i := 0; WHILE i < COUNT_LOGIC_TS DO
	iecDB_ts[ADRBASE_TS_LOGICAL + i].siq.b.SPI := sys_logic_ts[i];
	i := i + 1;
END_WHILE

i := 0; WHILE i < COUNT_VALVE DO
	iecDB_ts[ADRBASE_TS_VALVE + i*14 + 0].siq.b.SPI := sys_valve[i].flags.mode_dist;
	iecDB_ts[ADRBASE_TS_VALVE + i*14 + 1].siq.b.SPI := sys_valve[i].flags.mode_auto;
	iecDB_ts[ADRBASE_TS_VALVE + i*14 + 2].siq.b.SPI := sys_valve[i].flags.mode_imit;
	iecDB_ts[ADRBASE_TS_VALVE + i*14 + 3].siq.b.SPI := sys_valve[i].flags.mode_block;
	iecDB_ts[ADRBASE_TS_VALVE + i*14 + 4].siq.b.SPI := sys_valve[i].flags.cv_ok;
	iecDB_ts[ADRBASE_TS_VALVE + i*14 + 5].siq.b.SPI := sys_valve[i].flags.cv_fail;
	iecDB_ts[ADRBASE_TS_VALVE + i*14 + 6].siq.b.SPI := sys_valve[i].flags.fail_local;
	iecDB_ts[ADRBASE_TS_VALVE + i*14 + 7].siq.b.SPI := sys_valve[i].flags.fail_block;
	iecDB_ts[ADRBASE_TS_VALVE + i*14 + 8].siq.b.SPI := sys_valve[i].flags.fail_sm;
	iecDB_ts[ADRBASE_TS_VALVE + i*14 + 9].siq.b.SPI := sys_valve[i].flags.fail_start_open;
	iecDB_ts[ADRBASE_TS_VALVE + i*14 + 10].siq.b.SPI := sys_valve[i].flags.fail_open;
	iecDB_ts[ADRBASE_TS_VALVE + i*14 + 11].siq.b.SPI := sys_valve[i].flags.fail_start_close;
	iecDB_ts[ADRBASE_TS_VALVE + i*14 + 12].siq.b.SPI := sys_valve[i].flags.fail_close;
	iecDB_ts[ADRBASE_TS_VALVE + i*14 + 13].siq.b.SPI := sys_valve[i].flags.fail_moving;
	i := i + 1;
END_WHILE

i := 0; WHILE i < COUNT_STOP DO
	iecDB_ts[ADRBASE_TS_STOP + i*6 + 0].siq.b.SPI := sys_stop[i].flags.mode_block;
	iecDB_ts[ADRBASE_TS_STOP + i*6 + 1].siq.b.SPI := sys_stop[i].flags.msg_confirm;
	iecDB_ts[ADRBASE_TS_STOP + i*6 + 2].siq.b.SPI := sys_stop[i].flags.executing;
	iecDB_ts[ADRBASE_TS_STOP + i*6 + 3].siq.b.SPI := sys_stop[i].flags.done;
	iecDB_ts[ADRBASE_TS_STOP + i*6 + 4].siq.b.SPI := sys_stop[i].flags.fail;
	iecDB_ts[ADRBASE_TS_STOP + i*6 + 5].siq.b.SPI := sys_stop[i].flags.fail_block;
	i := i + 1;
END_WHILE

i := 0; WHILE i < COUNT_UNIT DO
	iecDB_ts[ADRBASE_TS_UNIT + i*10 + 0].siq.b.SPI := sys_unit[i].flags.mode_dist;
	iecDB_ts[ADRBASE_TS_UNIT + i*10 + 1].siq.b.SPI := sys_unit[i].flags.mode_auto;
	iecDB_ts[ADRBASE_TS_UNIT + i*10 + 2].siq.b.SPI := sys_unit[i].flags.mode_imit;
	iecDB_ts[ADRBASE_TS_UNIT + i*10 + 3].siq.b.SPI := sys_unit[i].flags.mode_block;
	iecDB_ts[ADRBASE_TS_UNIT + i*10 + 4].siq.b.SPI := sys_unit[i].flags.mode_work;
	iecDB_ts[ADRBASE_TS_UNIT + i*10 + 5].siq.b.SPI := sys_unit[i].flags.cv_ok;
	iecDB_ts[ADRBASE_TS_UNIT + i*10 + 6].siq.b.SPI := sys_unit[i].flags.cv_fail;	
	iecDB_ts[ADRBASE_TS_UNIT + i*10 + 7].siq.b.SPI := sys_unit[i].flags.fail_local;
	iecDB_ts[ADRBASE_TS_UNIT + i*10 + 8].siq.b.SPI := sys_unit[i].flags.fail_block;
	iecDB_ts[ADRBASE_TS_UNIT + i*10 + 9].siq.b.SPI := sys_unit[i].flags.fail_switch;
	i := i + 1;
END_WHILE

i := 0; WHILE i < COUNT_FAIL DO
	iecDB_ts[ADRBASE_TS_FAIL + i*3 + 0].siq.b.SPI := sys_fail[i].processed;
	iecDB_ts[ADRBASE_TS_FAIL + i*3 + 1].siq.b.SPI := sys_fail[i].block;
	iecDB_ts[ADRBASE_TS_FAIL + i*3 + 2].siq.b.SPI := sys_fail[i].imit;
	i := i + 1;
END_WHILE

i := 0; WHILE i < COUNT_WARN DO
	iecDB_ts[ADRBASE_TS_WARN + i*3 + 0].siq.b.SPI := sys_warn[i].processed;
	iecDB_ts[ADRBASE_TS_WARN + i*3 + 1].siq.b.SPI := sys_warn[i].block;
	iecDB_ts[ADRBASE_TS_WARN + i*3 + 2].siq.b.SPI := sys_warn[i].imit;
	i := i + 1;
END_WHILE

// ========== IEC_M_ME_TE
i := 0; WHILE i < COUNT_LOGIC_TE DO
	iecDB_te[ADRBASE_TE_LOGICAL + i].value := INT_TO_WORD(sys_logic_te[i]);
	iecDB_te[ADRBASE_TE_LOGICAL + i].qds.value := USINT_TO_BYTE(RLTBIO.Constants.QDS_STT_OK);
	i := i + 1;
END_WHILE

i := 0; WHILE i < COUNT_VALVE DO
	iecDB_te[ADRBASE_TE_VALVE + i*5 + 0].value := INT_TO_WORD(sys_valve[i].v_mode);
	iecDB_te[ADRBASE_TE_VALVE + i*5 + 0].qds.value := USINT_TO_BYTE(RLTBIO.Constants.QDS_STT_OK);
	iecDB_te[ADRBASE_TE_VALVE + i*5 + 1].value := INT_TO_WORD(sys_valve[i].v_state);
	iecDB_te[ADRBASE_TE_VALVE + i*5 + 1].qds.value := USINT_TO_BYTE(RLTBIO.Constants.QDS_STT_OK);
	iecDB_te[ADRBASE_TE_VALVE + i*5 + 2].value := sys_valve[i].sp.start;
	iecDB_te[ADRBASE_TE_VALVE + i*5 + 2].qds.value := USINT_TO_BYTE(RLTBIO.Constants.QDS_STT_OK);
	iecDB_te[ADRBASE_TE_VALVE + i*5 + 3].value := sys_valve[i].sp.moving;
	iecDB_te[ADRBASE_TE_VALVE + i*5 + 3].qds.value := USINT_TO_BYTE(RLTBIO.Constants.QDS_STT_OK);
	iecDB_te[ADRBASE_TE_VALVE + i*5 + 4].value := sys_valve[i].sp.press;
	iecDB_te[ADRBASE_TE_VALVE + i*5 + 4].qds.value := USINT_TO_BYTE(RLTBIO.Constants.QDS_STT_OK);
	i := i + 1;
END_WHILE

i := 0; WHILE i < COUNT_STOP DO
	iecDB_te[ADRBASE_TE_STOP + i*2 + 0].value := INT_TO_WORD(sys_stop[i].status);
	iecDB_te[ADRBASE_TE_STOP + i*2 + 0].qds.value := USINT_TO_BYTE(RLTBIO.Constants.QDS_STT_OK);
	iecDB_te[ADRBASE_TE_STOP + i*2 + 1].value := sys_stop[i].step;
	iecDB_te[ADRBASE_TE_STOP + i*2 + 1].qds.value := USINT_TO_BYTE(RLTBIO.Constants.QDS_STT_OK);
	i := i + 1;
END_WHILE

i := 0; WHILE i < COUNT_UNIT DO
	iecDB_te[ADRBASE_TE_UNIT + i*2 + 0].value := sys_unit[i].sp.switch;
	iecDB_te[ADRBASE_TE_UNIT + i*2 + 0].qds.value := USINT_TO_BYTE(RLTBIO.Constants.QDS_STT_OK);
	iecDB_te[ADRBASE_TE_UNIT + i*2 + 1].value := sys_unit[i].sp.work;
	iecDB_te[ADRBASE_TE_UNIT + i*2 + 1].qds.value := USINT_TO_BYTE(RLTBIO.Constants.QDS_STT_OK);
	i := i + 1;
END_WHILE

// ========== IEC_M_ME_TF
i := 0; WHILE i < COUNT_LOGIC_TF DO
	iecDB_tf[ADRBASE_TF_LOGICAL + i].value := sys_logic_tf[i];
	iecDB_tf[ADRBASE_TF_LOGICAL + i].qds.value := USINT_TO_BYTE(RLTBIO.Constants.QDS_STT_OK);
	i := i + 1;
END_WHILE

i := 0; WHILE i < COUNT_AI DO
	iecDB_tf[ADRBASE_TF_TI_VALUE + i*9 + 0].value := sys_ai[i].rTI;
	iecDB_tf[ADRBASE_TF_TI_VALUE + i*9 + 0].qds.value := USINT_TO_BYTE(sys_ai[i].qds);
	iecDB_tf[ADRBASE_TF_TI_VALUE + i*9 + 1].value := sys_ai[i].out_min;
	iecDB_tf[ADRBASE_TF_TI_VALUE + i*9 + 1].qds.value := USINT_TO_BYTE(RLTBIO.Constants.QDS_STT_OK);
	iecDB_tf[ADRBASE_TF_TI_VALUE + i*9 + 2].value := sys_ai[i].out_max;
	iecDB_tf[ADRBASE_TF_TI_VALUE + i*9 + 2].qds.value := USINT_TO_BYTE(RLTBIO.Constants.QDS_STT_OK);
	iecDB_tf[ADRBASE_TF_TI_VALUE + i*9 + 3].value := sys_ai[i].delta;
	iecDB_tf[ADRBASE_TF_TI_VALUE + i*9 + 3].qds.value := USINT_TO_BYTE(RLTBIO.Constants.QDS_STT_OK);
	iecDB_tf[ADRBASE_TF_TI_VALUE + i*9 + 4].value := sys_ai[i].val_fail_min;
	iecDB_tf[ADRBASE_TF_TI_VALUE + i*9 + 4].qds.value := USINT_TO_BYTE(RLTBIO.Constants.QDS_STT_OK);
	iecDB_tf[ADRBASE_TF_TI_VALUE + i*9 + 5].value := sys_ai[i].val_fail_max;
	iecDB_tf[ADRBASE_TF_TI_VALUE + i*9 + 5].qds.value := USINT_TO_BYTE(RLTBIO.Constants.QDS_STT_OK);
	iecDB_tf[ADRBASE_TF_TI_VALUE + i*9 + 6].value := sys_ai[i].val_warn_min;
	iecDB_tf[ADRBASE_TF_TI_VALUE + i*9 + 6].qds.value := USINT_TO_BYTE(RLTBIO.Constants.QDS_STT_OK);
	iecDB_tf[ADRBASE_TF_TI_VALUE + i*9 + 7].value := sys_ai[i].val_warn_max;
	iecDB_tf[ADRBASE_TF_TI_VALUE + i*9 + 7].qds.value := USINT_TO_BYTE(RLTBIO.Constants.QDS_STT_OK);
	iecDB_tf[ADRBASE_TF_TI_VALUE + i*9 + 8].value := sys_ai[i].hyst;
	iecDB_tf[ADRBASE_TF_TI_VALUE + i*9 + 8].qds.value := USINT_TO_BYTE(RLTBIO.Constants.QDS_STT_OK);
	i := i + 1;
END_WHILE

i := 0; WHILE i < COUNT_AO DO
	iecDB_tf[ADRBASE_TF_TR_VALUE + i*3 + 0].value := sys_ao[i].tr;
	iecDB_tf[ADRBASE_TF_TR_VALUE + i*3 + 0].qds.value := USINT_TO_BYTE(RLTBIO.Constants.QDS_STT_OK);
	iecDB_tf[ADRBASE_TF_TR_VALUE + i*3 + 1].value := sys_ao[i].in_min;
	iecDB_tf[ADRBASE_TF_TR_VALUE + i*3 + 1].qds.value := USINT_TO_BYTE(RLTBIO.Constants.QDS_STT_OK);
	iecDB_tf[ADRBASE_TF_TR_VALUE + i*3 + 2].value := sys_ao[i].in_max;
	iecDB_tf[ADRBASE_TF_TR_VALUE + i*3 + 2].qds.value := USINT_TO_BYTE(RLTBIO.Constants.QDS_STT_OK);
	i := i + 1;
END_WHILE

//========== C_SC_NA_1		через ИЛИ потому что могут быть и другие источники команд!
station.cmd.mode_auto_off := station.cmd.mode_auto_off OR		iecDB_tu[1];	iecDB_tu[1] := FALSE;
station.cmd.mode_auto_on := station.cmd.mode_auto_on OR			iecDB_tu[2];	iecDB_tu[2] := FALSE;
station.cmd.ack_control := station.cmd.ack_control OR			iecDB_tu[3];	iecDB_tu[3] := FALSE;
station.cmd.ack_valves := station.cmd.ack_valves OR				iecDB_tu[4];	iecDB_tu[4] := FALSE;
station.cmd.ack_units := station.cmd.ack_units OR				iecDB_tu[5];	iecDB_tu[5] := FALSE;
station.cmd.ack_alarms := station.cmd.ack_alarms OR				iecDB_tu[6];	iecDB_tu[6] := FALSE;
station.cmd.reset_imit := station.cmd.reset_imit OR 			iecDB_tu[7];	iecDB_tu[7] := FALSE;
station.cmd.imit_valves_on := station.cmd.imit_valves_on OR 	iecDB_tu[8];	iecDB_tu[8] := FALSE;
station.cmd.imit_valves_off := station.cmd.imit_valves_off OR	iecDB_tu[9];	iecDB_tu[9] := FALSE;
station.cmd.imit_units_on := station.cmd.imit_units_on OR		iecDB_tu[10];	iecDB_tu[10] := FALSE;
station.cmd.imit_units_off := station.cmd.imit_units_off OR		iecDB_tu[11];	iecDB_tu[11] := FALSE;
station.cmd.block_sound_on := station.cmd.block_sound_on OR		iecDB_tu[12];	iecDB_tu[12] := FALSE;
station.cmd.block_sound_off := station.cmd.block_sound_off OR	iecDB_tu[13];	iecDB_tu[13] := FALSE;
station.cmd.sound_on := station.cmd.sound_on OR					iecDB_tu[14];	iecDB_tu[14] := FALSE;
station.cmd.sound_off := station.cmd.sound_off OR				iecDB_tu[15];	iecDB_tu[15] := FALSE;
station.cmd.alarm_on := station.cmd.alarm_on OR					iecDB_tu[16];	iecDB_tu[16] := FALSE;
station.cmd.alarm_off := station.cmd.alarm_off OR				iecDB_tu[17];	iecDB_tu[17] := FALSE;
station.cmd.lamps_on := station.cmd.lamps_on OR 				iecDB_tu[18];	iecDB_tu[18] := FALSE;
station.cmd.lamps_off := station.cmd.lamps_off OR 				iecDB_tu[19];	iecDB_tu[19] := FALSE;
//i := 0; WHILE i < COUNT_LOGIC_CMD DO
//	iecDB_tu[ADRBASE_CMD_LOGIC + i] := FALSE;
//	i := i + 1;
//END_WHILE

i := 0; WHILE i < COUNT_VALVE DO
	IF station.mode <> en_stt_mode.MODE_AUTO THEN
		sys_valve[i].cmd.open := sys_valve[i].cmd.open OR			iecDB_tu[ADRBASE_CMD_VALVE + i*8 + 0];
		sys_valve[i].cmd.close := sys_valve[i].cmd.close OR			iecDB_tu[ADRBASE_CMD_VALVE + i*8 + 1];
		sys_valve[i].cmd.stop := sys_valve[i].cmd.stop OR			iecDB_tu[ADRBASE_CMD_VALVE + i*8 + 2];
	ELSE
		IF sys_valve[i].cmd.open OR sys_valve[i].cmd.close OR sys_valve[i].cmd.stop THEN
			station.fail_control := TRUE;
		END_IF
	END_IF
	iecDB_tu[ADRBASE_CMD_VALVE + i*8 + 0] := FALSE;
	iecDB_tu[ADRBASE_CMD_VALVE + i*8 + 1] := FALSE;
	iecDB_tu[ADRBASE_CMD_VALVE + i*8 + 2] := FALSE;
	sys_valve[i].cmd.ack := sys_valve[i].cmd.ack OR				iecDB_tu[ADRBASE_CMD_VALVE + i*8 + 3];		iecDB_tu[ADRBASE_CMD_VALVE + i*8 + 3] := FALSE;
	sys_valve[i].cmd.imit_on := sys_valve[i].cmd.imit_on OR		iecDB_tu[ADRBASE_CMD_VALVE + i*8 + 4];		iecDB_tu[ADRBASE_CMD_VALVE + i*8 + 4] := FALSE;
	sys_valve[i].cmd.imit_off := sys_valve[i].cmd.imit_off OR	iecDB_tu[ADRBASE_CMD_VALVE + i*8 + 5];		iecDB_tu[ADRBASE_CMD_VALVE + i*8 + 5] := FALSE;
	sys_valve[i].cmd.block_on := sys_valve[i].cmd.block_on OR	iecDB_tu[ADRBASE_CMD_VALVE + i*8 + 6];		iecDB_tu[ADRBASE_CMD_VALVE + i*8 + 6] := FALSE;
	sys_valve[i].cmd.block_off := sys_valve[i].cmd.block_off OR	iecDB_tu[ADRBASE_CMD_VALVE + i*8 + 7];		iecDB_tu[ADRBASE_CMD_VALVE + i*8 + 7] := FALSE;
	i := i + 1;
END_WHILE

i := 0; WHILE i < COUNT_STOP DO
	sys_stop[i].cmd.ack := sys_stop[i].cmd.ack OR				iecDB_tu[ADRBASE_CMD_STOP + i*6 + 0];		iecDB_tu[ADRBASE_CMD_STOP + i*6 + 0] := FALSE;
	sys_stop[i].cmd.block_on := sys_stop[i].cmd.block_on OR 	iecDB_tu[ADRBASE_CMD_STOP + i*6 + 1];		iecDB_tu[ADRBASE_CMD_STOP + i*6 + 1] := FALSE;
	sys_stop[i].cmd.block_off := sys_stop[i].cmd.block_off OR	iecDB_tu[ADRBASE_CMD_STOP + i*6 + 2];		iecDB_tu[ADRBASE_CMD_STOP + i*6 + 2] := FALSE;
	sys_stop[i].cmd.execute := sys_stop[i].cmd.execute OR		iecDB_tu[ADRBASE_CMD_STOP + i*6 + 3];		iecDB_tu[ADRBASE_CMD_STOP + i*6 + 3] := FALSE;
	sys_stop[i].cmd.confirm := sys_stop[i].cmd.confirm OR 		iecDB_tu[ADRBASE_CMD_STOP + i*6 + 4];		iecDB_tu[ADRBASE_CMD_STOP + i*6 + 4] := FALSE;
	sys_stop[i].cmd.reject := sys_stop[i].cmd.reject OR 		iecDB_tu[ADRBASE_CMD_STOP + i*6 + 5];		iecDB_tu[ADRBASE_CMD_STOP + i*6 + 5] := FALSE;
	i := i + 1;
END_WHILE

i := 0; WHILE i < COUNT_UNIT DO
	IF station.mode <> en_stt_mode.MODE_AUTO THEN
		sys_unit[i].cmd.on := sys_unit[i].cmd.on OR 				iecDB_tu[ADRBASE_CMD_UNIT + i*7 + 0];
		sys_unit[i].cmd.off := sys_unit[i].cmd.off OR 				iecDB_tu[ADRBASE_CMD_UNIT + i*7 + 1];
	ELSE
		IF sys_unit[i].cmd.on OR sys_unit[i].cmd.off THEN
			station.fail_control := TRUE;
		END_IF
	END_IF
	iecDB_tu[ADRBASE_CMD_UNIT + i*7 + 0] := FALSE;
	iecDB_tu[ADRBASE_CMD_UNIT + i*7 + 1] := FALSE;
	sys_unit[i].cmd.ack := sys_unit[i].cmd.ack OR 				iecDB_tu[ADRBASE_CMD_UNIT + i*7 + 2];		iecDB_tu[ADRBASE_CMD_UNIT + i*7 + 2] := FALSE;
	sys_unit[i].cmd.imit_on := sys_unit[i].cmd.imit_on OR 		iecDB_tu[ADRBASE_CMD_UNIT + i*7 + 3];		iecDB_tu[ADRBASE_CMD_UNIT + i*7 + 3] := FALSE;
	sys_unit[i].cmd.imit_off := sys_unit[i].cmd.imit_off OR 	iecDB_tu[ADRBASE_CMD_UNIT + i*7 + 4];		iecDB_tu[ADRBASE_CMD_UNIT + i*7 + 4] := FALSE;
	sys_unit[i].cmd.block_on := sys_unit[i].cmd.block_on OR 	iecDB_tu[ADRBASE_CMD_UNIT + i*7 + 5];		iecDB_tu[ADRBASE_CMD_UNIT + i*7 + 5] := FALSE;
	sys_unit[i].cmd.block_off := sys_unit[i].cmd.block_off OR	iecDB_tu[ADRBASE_CMD_UNIT + i*7 + 6];		iecDB_tu[ADRBASE_CMD_UNIT + i*7 + 6] := FALSE;
	i := i + 1;
END_WHILE

i := 0; WHILE i < COUNT_FAIL DO
	sys_fail[i].cmd_ack := sys_fail[i].cmd_ack OR iecDB_tu[ADRBASE_CMD_FAIL + i*5 + 0];		iecDB_tu[ADRBASE_CMD_FAIL + i*5 + 0] := FALSE;
	IF iecDB_tu[ADRBASE_CMD_FAIL + i*5 + 1] THEN
		sys_fail[i].block := TRUE;										iecDB_tu[ADRBASE_CMD_FAIL + i*5 + 1] := FALSE;
	END_IF
	IF iecDB_tu[ADRBASE_CMD_FAIL + i*5 + 2] THEN
		sys_fail[i].block := FALSE;										iecDB_tu[ADRBASE_CMD_FAIL + i*5 + 2] := FALSE;
	END_IF
	IF sys_fail_m[i].sp.b <> sys_fail[i].block THEN
		sys_fail_m[i].sp0.b := sys_fail[i].block;
		sys_fail_m[i].cmd := TRUE;
	END_IF
	IF iecDB_tu[ADRBASE_CMD_FAIL + i*5 + 3] THEN
		sys_fail[i].imit := TRUE;										iecDB_tu[ADRBASE_CMD_FAIL + i*5 + 3] := FALSE;
	END_IF
	IF iecDB_tu[ADRBASE_CMD_FAIL + i*5 + 4] THEN
		sys_fail[i].imit := FALSE;										iecDB_tu[ADRBASE_CMD_FAIL + i*5 + 4] := FALSE;
	END_IF
	i := i + 1;
END_WHILE

i := 0; WHILE i < COUNT_WARN DO
	IF iecDB_tu[ADRBASE_CMD_WARN + i*4 + 0] THEN
		sys_warn[i].block := TRUE;										iecDB_tu[ADRBASE_CMD_WARN + i*4 + 0] := FALSE;
	END_IF
	IF iecDB_tu[ADRBASE_CMD_WARN + i*4 + 1] THEN
		sys_warn[i].block := FALSE;										iecDB_tu[ADRBASE_CMD_WARN + i*4 + 1] := FALSE;
	END_IF
	IF sys_warn_m[i].sp.b <> sys_warn[i].block THEN
		sys_warn_m[i].sp0.b := sys_warn[i].block;
		sys_warn_m[i].cmd := TRUE;
	END_IF
	IF iecDB_tu[ADRBASE_CMD_WARN + i*4 + 2] THEN
		sys_warn[i].imit := TRUE;										iecDB_tu[ADRBASE_CMD_WARN + i*4 + 2] := FALSE;
	END_IF
	IF iecDB_tu[ADRBASE_CMD_WARN + i*4 + 3] THEN
		sys_warn[i].imit := FALSE;										iecDB_tu[ADRBASE_CMD_WARN + i*4 + 3] := FALSE;
	END_IF
	i := i + 1;
END_WHILE

//========== IEC_C_SE_NB
//logic

i := 0; WHILE i < COUNT_VALVE DO
	sys_valve_sp[i*3 + 0].sp0.ui := iecDB_tri[ADRBASE_NB_VALVE + i*3 + 0];
	sys_valve_sp[i*3 + 0].cmd := sys_valve_sp[i*3 + 0].cmd OR iecDB_tri_act[ADRBASE_NB_VALVE + i*3 + 0];
	iecDB_tri_act[ADRBASE_NB_VALVE + i*3 + 0] := FALSE;
	sys_valve_sp[i*3 + 1].sp0.ui := iecDB_tri[ADRBASE_NB_VALVE + i*3 + 1];
	sys_valve_sp[i*3 + 1].cmd := sys_valve_sp[i*3 + 1].cmd OR iecDB_tri_act[ADRBASE_NB_VALVE + i*3 + 1];
	iecDB_tri_act[ADRBASE_NB_VALVE + i*3 + 1] := FALSE;
	sys_valve_sp[i*3 + 2].sp0.ui := iecDB_tri[ADRBASE_NB_VALVE + i*3 + 2];
	sys_valve_sp[i*3 + 2].cmd := sys_valve_sp[i*3 + 2].cmd OR iecDB_tri_act[ADRBASE_NB_VALVE + i*3 + 2];
	iecDB_tri_act[ADRBASE_NB_VALVE + i*3 + 2] := FALSE;
	i := i + 1;
END_WHILE

i := 0; WHILE i < COUNT_UNIT DO
	sys_unit_sp[i*2 + 0].sp0.ui := iecDB_tri[ADRBASE_NB_UNIT + i*2 + 0];
	sys_unit_sp[i*2 + 0].cmd := sys_unit_sp[i*2 + 0].cmd OR iecDB_tri_act[ADRBASE_NB_UNIT + i*2 + 0];
	iecDB_tri_act[ADRBASE_NB_UNIT + i*2 + 0] := FALSE;
	sys_unit_sp[i*2 + 1].sp0.ui := iecDB_tri[ADRBASE_NB_UNIT + i*2 + 1];
	sys_unit_sp[i*2 + 1].cmd := sys_unit_sp[i*2 + 1].cmd OR iecDB_tri_act[ADRBASE_NB_UNIT + i*2 + 1];
	iecDB_tri_act[ADRBASE_NB_UNIT + i*2 + 1] := FALSE;
	i := i + 1;
END_WHILE

//========== IEC_C_SE_NC
//logic

i := 0; WHILE i < COUNT_AI DO
	sys_ai_sp[i*8 + 0].sp0.re := iecDB_trf[ADRBASE_NC_TI + i*8 + 0];
	sys_ai_sp[i*8 + 0].cmd := sys_ai_sp[i*8 + 0].cmd OR iecDB_trf_act[ADRBASE_NC_TI + i*8 + 0];
	iecDB_trf_act[ADRBASE_NC_TI + i*8 + 0] := FALSE;
	sys_ai_sp[i*8 + 1].sp0.re := iecDB_trf[ADRBASE_NC_TI + i*8 + 1];
	sys_ai_sp[i*8 + 1].cmd := sys_ai_sp[i*8 + 1].cmd OR iecDB_trf_act[ADRBASE_NC_TI + i*8 + 1];
	iecDB_trf_act[ADRBASE_NC_TI + i*8 + 1] := FALSE;
	sys_ai_sp[i*8 + 2].sp0.re := iecDB_trf[ADRBASE_NC_TI + i*8 + 2];
	sys_ai_sp[i*8 + 2].cmd := sys_ai_sp[i*8 + 2].cmd OR iecDB_trf_act[ADRBASE_NC_TI + i*8 + 2];
	iecDB_trf_act[ADRBASE_NC_TI + i*8 + 2] := FALSE;
	sys_ai_sp[i*8 + 3].sp0.re := iecDB_trf[ADRBASE_NC_TI + i*8 + 3];
	sys_ai_sp[i*8 + 3].cmd := sys_ai_sp[i*8 + 3].cmd OR iecDB_trf_act[ADRBASE_NC_TI + i*8 + 3];
	iecDB_trf_act[ADRBASE_NC_TI + i*8 + 3] := FALSE;
	sys_ai_sp[i*8 + 4].sp0.re := iecDB_trf[ADRBASE_NC_TI + i*8 + 4];
	sys_ai_sp[i*8 + 4].cmd := sys_ai_sp[i*8 + 4].cmd OR iecDB_trf_act[ADRBASE_NC_TI + i*8 + 4];
	iecDB_trf_act[ADRBASE_NC_TI + i*8 + 4] := FALSE;
	sys_ai_sp[i*8 + 5].sp0.re := iecDB_trf[ADRBASE_NC_TI + i*8 + 5];
	sys_ai_sp[i*8 + 5].cmd := sys_ai_sp[i*8 + 5].cmd OR iecDB_trf_act[ADRBASE_NC_TI + i*8 + 5];
	iecDB_trf_act[ADRBASE_NC_TI + i*8 + 5] := FALSE;
	sys_ai_sp[i*8 + 6].sp0.re := iecDB_trf[ADRBASE_NC_TI + i*8 + 6];
	sys_ai_sp[i*8 + 6].cmd := sys_ai_sp[i*8 + 6].cmd OR iecDB_trf_act[ADRBASE_NC_TI + i*8 + 6];
	iecDB_trf_act[ADRBASE_NC_TI + i*8 + 6] := FALSE;
	sys_ai_sp[i*8 + 7].sp0.re := iecDB_trf[ADRBASE_NC_TI + i*8 + 7];
	sys_ai_sp[i*8 + 7].cmd := sys_ai_sp[i*8 + 7].cmd OR iecDB_trf_act[ADRBASE_NC_TI + i*8 + 7];
	iecDB_trf_act[ADRBASE_NC_TI + i*8 + 7] := FALSE;	
	i := i + 1;
END_WHILE

i := 0; WHILE i < COUNT_AO DO
	sys_ao_sp[i*3 + 0].sp0.re := iecDB_trf[ADRBASE_NC_TR + i*3 + 0];
	sys_ao_sp[i*3 + 0].cmd := sys_ao_sp[i*3 + 0].cmd OR iecDB_trf_act[ADRBASE_NC_TR + i*3 + 0];
	iecDB_trf_act[ADRBASE_NC_TR + i*3 + 0] := FALSE;
	sys_ao_sp[i*3 + 1].sp0.re := iecDB_trf[ADRBASE_NC_TR + i*3 + 1];
	sys_ao_sp[i*3 + 1].cmd := sys_ao_sp[i*3 + 1].cmd OR iecDB_trf_act[ADRBASE_NC_TR + i*3 + 1];
	iecDB_trf_act[ADRBASE_NC_TR + i*3 + 1] := FALSE;
	sys_ao_sp[i*3 + 2].sp0.re := iecDB_trf[ADRBASE_NC_TR + i*3 + 2];
	sys_ao_sp[i*3 + 2].cmd := sys_ao_sp[i*3 + 2].cmd OR iecDB_trf_act[ADRBASE_NC_TR + i*3 + 2];
	iecDB_trf_act[ADRBASE_NC_TR + i*3 + 2] := FALSE;
	i := i + 1;
END_WHILE
END_METHOD

METHOD Cyclic_Station
VAR_INPUT
END_VAR
VAR
	res: SysTimeRtc.SysTypes.RTS_IEC_RESULT;
	i, c: UINT;
END_VAR
//init
//init^

res := SysTimeRtc.SysTimeRtcHighResGet(station.time_sys);
res := SysTimeRtc.SysTimeRtcConvertHighResToLocal(station.time_sys, station.time_plc);

IF station.cfg.conf_valve_dist THEN
	//station.di_valve_dist := sys_di[station.num_di_valve_dist].ts;
	IF NOT sys_di[station.num_di_valve_dist].ts THEN
		station.mode := en_stt_mode.MODE_BUTTON;
	ELSIF station.mode_auto THEN
		station.mode := en_stt_mode.MODE_AUTO;
	ELSE
		station.mode := en_stt_mode.MODE_MANUAL;
	END_IF
ELSE
	//station.di_valve_dist := FALSE;
	c := 0;
	i := 0; WHILE i < COUNT_VALVE DO
		IF sys_valve[i].v_mode = RLTAB.en_valve_mode.MODE_BUTTON OR sys_valve[i].v_mode = RLTAB.en_valve_mode.MODE_NONE THEN
			c := c + 1;
		END_IF
		i := i + 1;
	END_WHILE
	IF c = COUNT_VALVE THEN
		station.mode := en_stt_mode.MODE_BUTTON;
	ELSIF c > 0 THEN
		station.mode := en_stt_mode.MODE_PART_BUTTON;
	ELSIF station.mode_auto THEN
		station.mode := en_stt_mode.MODE_AUTO;
	ELSE
		station.mode := en_stt_mode.MODE_MANUAL;
	END_IF
END_IF
IF station.cfg.conf_valve_cv THEN
	//station.di_valve_cv := sys_di[station.num_di_valve_cv].ts;
	station.do_valve_cv := FALSE;
	i := 0; WHILE i < COUNT_VALVE DO
		station.do_valve_cv := station.do_valve_cv OR sys_valve[i].out.do_cv;
		i := i + 1;
	END_WHILE
	sys_do[station.num_do_valve_cv].cmd_on := station.do_valve_cv;
ELSE
	// запоняется в Cyclic_Out
	station.do_valve_cv := FALSE;
END_IF
(* temp unused
IF station.cfg.conf_unit_dist THEN
	//station.di_unit_dist := sys_di[station.num_di_unit_dist].ts;
	//TO DO
ELSE
	//station.di_unit_dist := FALSE;
END_IF
IF station.cfg.conf_unit_cv THEN
	//station.di_unit_cv := sys_di[station.num_di_unit_cv].ts;
	//TO DO
ELSE
	//station.di_unit_cv := FALSE;
END_IF
*)
IF station.cfg.conf_ack THEN
	station.di_ack := sys_di[station.num_di_ack].ts;
	station.r_ack(CLK := station.di_ack);
	//IF station.r_ack.Q THEN
	//END_IF
ELSE
	station.di_ack := FALSE;
END_IF
IF station.cfg.conf_stop_1 THEN
	station.di_stop_1 := sys_di[station.num_di_stop_1].ts;
	station.r_stop_1(CLK := station.di_stop_1);
	IF station.r_stop_1.Q THEN
		IF station.mode > en_stt_mode.MODE_PART_BUTTON THEN
			sys_stop[station.num_stop_1].cmd.execute := TRUE;
			station.stop_impossible := FALSE;
		ELSE
			station.stop_impossible := TRUE;
		END_IF
	END_IF
ELSE
	station.di_stop_1 := FALSE;
END_IF
IF station.cfg.conf_stop_2 THEN
	station.di_stop_2 := sys_di[station.num_di_stop_2].ts;
	station.r_stop_2(CLK := station.di_stop_2);
	IF station.r_stop_2.Q THEN
		IF station.mode > en_stt_mode.MODE_PART_BUTTON THEN
			sys_stop[station.num_stop_2].cmd.execute := TRUE;
			station.stop_impossible := FALSE;
		ELSE
			station.stop_impossible := TRUE;
		END_IF
	END_IF
ELSE
	station.di_stop_2 := FALSE;
END_IF

IF station.cfg.conf_test_sound THEN
	station.di_sound := sys_di[station.num_di_sound].ts;
ELSE
	station.di_sound := FALSE;
END_IF
IF station.cfg.conf_test_alarm THEN
	station.di_alarm := sys_di[station.num_di_alarm].ts;
ELSE
	station.di_alarm := FALSE;
END_IF
IF station.cfg.conf_lamps THEN
	station.di_lamps := sys_di[station.num_di_lamps].ts;
ELSE
	station.di_lamps := FALSE;
END_IF

IF (station.mode = en_stt_mode.MODE_BUTTON OR station.mode = en_stt_mode.MODE_PART_BUTTON) AND station.p_mode = en_stt_mode.MODE_AUTO THEN
	station.cmd.mode_auto_reset := TRUE;
END_IF
station.p_mode := station.mode;


IF station.cmd.mode_auto_off THEN		// 1	Перевести ГРС в автоматизированный режим
	station.cmd.mode_auto_off := FALSE;
	station.mode_auto := FALSE;
END_IF
IF station.cmd.mode_auto_on THEN		// 2	Перевести ГРС в автоматический режим
	station.cmd.mode_auto_on := FALSE;
	IF NOT station.auto_blocked THEN
		station.mode_auto := TRUE;
		station.auto_reset := FALSE;
	END_IF
END_IF
IF station.cmd.mode_auto_reset THEN		// technical
	station.cmd.mode_auto_reset := FALSE;
	station.mode_auto := FALSE;
	station.auto_reset := TRUE;
END_IF

IF station.cmd.ack_control THEN			// 3	Квитировать ошибку управления
	station.cmd.ack_control := FALSE;
	
	station.fail_control := FALSE;
	station.stop_impossible := FALSE;
	station.auto_reset := FALSE;
	i := 0; WHILE i < COUNT_SERVERS DO
		station.fail_center[i] := FALSE;
		i := i + 1;
	END_WHILE
END_IF
IF station.cmd.ack_valves THEN			// 4	Квитирование аварий задвижек
	station.cmd.ack_valves := FALSE;
	i := 0; WHILE i < COUNT_VALVE DO
		sys_valve[i].cmd.ack := TRUE;
		i := i + 1;
	END_WHILE
END_IF
IF station.cmd.ack_units THEN			// 5	Квитирование аварий вентиляторов и агрегатов 
	station.cmd.ack_units := FALSE;
	i := 0; WHILE i < COUNT_UNIT DO
		sys_unit[i].cmd.ack := TRUE;
		i := i + 1;
	END_WHILE
END_IF
IF station.cmd.ack_alarms OR station.r_ack.Q THEN	// 6	Квитирование аварий
	station.cmd.ack_alarms := FALSE;
	i := 0; WHILE i < COUNT_STOP DO
		sys_stop[i].cmd.ack := TRUE;
		i := i + 1;
	END_WHILE
	i := 0; WHILE i < COUNT_FAIL DO
		sys_fail[i].cmd_ack := TRUE;
		i := i + 1;
	END_WHILE
	station.do_sound := FALSE;
	station.do_alarm := FALSE;
	station.do_lamp_fail := FALSE;
	station.do_lamp_alarm := FALSE;
	station.do_lamp_fire := FALSE;
	station.do_lamp_gas := FALSE;
END_IF

IF station.cmd.reset_imit THEN			// 7	Сброс имитации сигнализации
	station.cmd.reset_imit := FALSE;
	i := 0; WHILE i < COUNT_FAIL DO
		sys_fail[i].imit := FALSE;
		i := i + 1;
	END_WHILE
	i := 0; WHILE i < COUNT_WARN DO
		sys_warn[i].imit := FALSE;
		i := i + 1;
	END_WHILE
END_IF
IF station.cmd.imit_valves_on THEN		// 8	Включить имитацию всех задвижек
	station.cmd.imit_valves_on := FALSE;
	IF station.mode < en_stt_mode.MODE_AUTO THEN
		i := 0; WHILE i < COUNT_VALVE DO
			sys_valve[i].cmd.imit_on := TRUE;
			i := i + 1;
		END_WHILE
	ELSE
		station.fail_control := TRUE;
	END_IF
END_IF
IF station.cmd.imit_valves_off THEN		// 9	Выключить имитацию всех задвижек
	station.cmd.imit_valves_off := FALSE;
	IF station.mode < en_stt_mode.MODE_AUTO THEN
		i := 0; WHILE i < COUNT_VALVE DO
			sys_valve[i].cmd.imit_off := TRUE;
			i := i + 1;
		END_WHILE
	ELSE
		station.fail_control := TRUE;
	END_IF
END_IF
IF station.cmd.imit_units_on THEN		// 10	Включить имитацию всех вентиляторов
	station.cmd.imit_units_on := FALSE;
	IF station.mode < en_stt_mode.MODE_AUTO THEN
		i := 0; WHILE i < COUNT_UNIT DO
			sys_unit[i].cmd.imit_on := TRUE;
			i := i + 1;
		END_WHILE
	ELSE
		station.fail_control := TRUE;
	END_IF
END_IF
IF station.cmd.imit_units_off THEN		// 11	Выключить имитацию всех вентиляторов
	station.cmd.imit_units_off := FALSE;
	IF station.mode < en_stt_mode.MODE_AUTO THEN
		i := 0; WHILE i < COUNT_UNIT DO
			sys_unit[i].cmd.imit_off := TRUE;
			i := i + 1;
		END_WHILE
	ELSE
		station.fail_control := TRUE;
	END_IF
END_IF

IF station.cmd.block_sound_on THEN		// 12	Включить блокировку звуковой сигнализации
	station.cmd.block_sound_on := FALSE;
	IF station.cfg.conf_sound_block THEN
		station.do_sound := FALSE;
		station.do_alarm := FALSE;
	ELSE
		station.fail_control := TRUE;	// отреагируем так чтобы операторы не тупили
	END_IF
END_IF
IF station.cmd.block_sound_off THEN		// 13	Выключить блокировку звуковой сигнализации
	station.cmd.block_sound_off := FALSE;
	station.sound_blocked := TRUE;
END_IF

IF station.cmd.sound_on THEN			// 14	Включить звонок
	station.cmd.sound_on := FALSE;
	station.do_sound := TRUE;
END_IF
IF station.cmd.sound_off THEN			// 15	Выключить звонок
	station.cmd.sound_off := FALSE;
	station.do_sound := FALSE;
END_IF
IF station.cmd.alarm_on THEN			// 16	Включить сирену
	station.cmd.alarm_on := FALSE;
	station.do_alarm := TRUE;
END_IF
IF station.cmd.alarm_off THEN			// 17	Выключить сирену
	station.cmd.alarm_off := FALSE;
	station.do_alarm := FALSE;
END_IF

IF station.cmd.lamps_on THEN			// 18	Включить тест ламп
	station.cmd.lamps_on := FALSE;
	station.do_lamps := TRUE;
END_IF
IF station.cmd.lamps_off THEN			// 19	Выключить тест ламп
	station.cmd.lamps_off := FALSE;
	station.do_lamps := FALSE;
END_IF

(* 	request_confirm: BOOL;
	request_reject: BOOL; *)

IF station.cfg.conf_sound THEN
	sys_do[station.num_do_sound].cmd_on := station.do_sound OR station.di_sound OR station.do_alarm;
ELSE
	station.do_sound := FALSE;
END_IF
IF station.cfg.conf_alarm THEN
	sys_do[station.num_do_alarm].cmd_on := station.do_alarm OR station.di_alarm OR (station.cfg.conf_warn_is_alarm AND station.do_sound);
ELSE
	station.do_alarm := FALSE;
END_IF

IF station.cfg.conf_warn THEN
	sys_do[station.num_do_lamp_alarm].cmd_on := station.do_lamp_alarm OR station.di_lamps OR station.do_lamps OR station.do_lamp_fail;
ELSE
	station.do_lamp_alarm := FALSE;
END_IF
IF station.cfg.conf_fail THEN
	sys_do[station.num_do_lamp_fail].cmd_on := station.do_lamp_fail OR station.di_lamps OR station.do_lamps;
ELSE
	station.do_lamp_fail := FALSE;
END_IF
IF station.cfg.conf_fire THEN
	sys_do[station.num_do_lamp_fire].cmd_on := station.do_lamp_fire OR station.di_lamps OR station.do_lamps;
ELSE
	station.do_lamp_fire := FALSE;
END_IF
IF station.cfg.conf_gas THEN
	sys_do[station.num_do_lamp_gas].cmd_on := station.do_lamp_gas OR station.di_lamps OR station.do_lamps;
ELSE
	station.do_lamp_gas := FALSE;
END_IF


sys_logic_ts[0] := station.global_imit_di;
sys_logic_ts[1] := station.global_imit_ai;
sys_logic_ts[2] := station.global_imit_do;
sys_logic_ts[3] := station.global_imit_ao;
IF station.cfg.conf_valve_cv THEN
	sys_logic_ts[4] := sys_valve[0].flags.cv_ok;
	sys_logic_ts[5] := station.fail_valve_cv;
ELSE
	sys_logic_ts[4] := FALSE;
	sys_logic_ts[5] := FALSE;
END_IF
IF station.cfg.conf_unit_cv THEN
	sys_logic_ts[6] := sys_unit[0].flags.cv_ok;;
	sys_logic_ts[7] := station.fail_unit_cv;
ELSE
	sys_logic_ts[6] := FALSE;
	sys_logic_ts[7] := FALSE;
END_IF
sys_logic_ts[8] := station.sound_blocked;
sys_logic_ts[9] := station.global_imit_valve;
sys_logic_ts[10] := station.global_imit_unit;
sys_logic_ts[11] := station.do_lamp_fail;
sys_logic_ts[12] := station.do_lamp_alarm;
sys_logic_ts[13] := station.global_stop;
sys_logic_ts[14] := station.stop_impossible;
sys_logic_ts[15] := station.auto_blocked; //user!
sys_logic_ts[16] := station.auto_reset;
sys_logic_ts[17] := station.fail_control;

sys_logic_te[0] := options.last_group;
sys_logic_te[1] := station.mode;
sys_logic_te[2] := station.user;
//...
sys_logic_te[18] := UINT_TO_INT(station.time_plc.wYear);
sys_logic_te[19] := UINT_TO_INT(station.time_plc.wMonth);
sys_logic_te[20] := UINT_TO_INT(station.time_plc.wDay);
sys_logic_te[21] := UINT_TO_INT(station.time_plc.wHour);
sys_logic_te[22] := UINT_TO_INT(station.time_plc.wMinute);
IF station.cfg.conf_out_seconds THEN
	sys_logic_te[23] := UINT_TO_INT(station.time_plc.wSecond);
END_IF


diag.err_cfg_servers := COUNT_MAX_SERVERS > RLTNU.IECDefines.IEC_CLIENT_MAX_COUNT;
diag.err_cfg_groups := COUNT_LINE_GROUPS = 0 OR COUNT_LINE_GROUPS >= COUNT_LINES;
diag.err_cfg_lines := COUNT_LINES < 2;

diag.ai_empty_size := (MAX_COUNT_AI - COUNT_AI) * 9;
END_METHOD

END_PROGRAM

// A1_01A/Application/App104
PROGRAM App104
VAR_INPUT
	enable: BOOL := 0;
	srv: RLTNU.IEC104Server; //VAR
END_VAR
VAR
	db: RLTNU.IECDB;
	
	ts: ARRAY[0..IEC_COUNT_M_SP_TB_1-1] OF RLTNU.IEC_M_SP_NA;
	ti: ARRAY[0..IEC_COUNT_M_ME_TE_1-1] OF RLTNU.IEC_M_ME_NB;
	tf: ARRAY[0..IEC_COUNT_M_ME_TF_1-1] OF RLTNU.IEC_M_ME_NC;
	event: RLTNU.IECSpontaneousEvent;
	command: RLTNU.IECCommand;
	
	tim: ULINT;
	state: UINT;
	i: UDINT;
END_VAR

IF NOT enable THEN
	RETURN;
END_IF

CASE state OF
	0:
		srv.activate := TRUE;
		
		//port
		//srv.commonASDUAddress := 1;
		//srv.windowSizeK := 12;
		//srv.windowSizeW := 8;
		//srv.timeoutK := T#30S;
		srv.startAddressTS := ADRBASE_IEC_M_SP_TB_1;
		srv.startAddressTI := ADRBASE_IEC_M_ME_TE_1;
		srv.startAddressTF := ADRBASE_IEC_M_ME_TF_1;
		srv.startAddressTU := ADRBASE_IEC_C_SC_NA_1;
		srv.startAddressTRI := ADRBASE_IEC_C_SE_NB_1;
		srv.startAddressTRF := ADRBASE_IEC_C_SE_NC_1;
		
		srv.commandMaxCount := 30000;
		srv.eventMaxCount := 30000;
		srv.inOutPacketMaxCount := 30000;
		
		db.ts := ADR(ts);
		db.ts_count := IEC_COUNT_M_SP_TB_1;
		db.ti := ADR(ti);
		db.ti_count := IEC_COUNT_M_ME_TE_1;
		db.tf := ADR(tf);
		db.tf_count := IEC_COUNT_M_ME_TF_1;
		db.tu_count := IEC_COUNT_C_SC_NA_1;
		db.tri_count := IEC_COUNT_C_SE_NB_1;
		db.trf_count := IEC_COUNT_C_SE_NC_1;
			
		srv.db := db;
		
		state := 10;
		
		FOR i := 0 TO IEC_COUNT_M_SP_TB_1-1 DO
			IF ts[i].siq.value <> iecDB_ts[i].siq.value THEN
				ts[i].siq.value := iecDB_ts[i].siq.value;
				
				RLTNU.SysTimeRtc.SysTimeRtcHighResGet(pTimestamp := tim);				
				event.addressObjectInformation := UDINT_TO_WORD(srv.startAddressTS + i);
				IF ts[i].siq.value.0 THEN event.value.ts := 1; ELSE event.value.ts := 0; END_IF
				event.qds.value := ts[i].siq.value;
				event.timeshtamp := tim;
				srv.setEvent(evt_type:= RLTNU.IECEventTypes.TS, event := event);
			END_IF
		END_FOR
		FOR i := 0 TO IEC_COUNT_M_ME_TE_1-1 DO
			IF ti[i].value <> iecDB_te[i].value OR ti[i].qds.value <> iecDB_te[i].qds.value THEN
				ti[i].value := iecDB_te[i].value;
				ti[i].qds.value := iecDB_te[i].qds.value;
				
				RLTNU.SysTimeRtc.SysTimeRtcHighResGet(pTimestamp := tim);				
				event.addressObjectInformation := UDINT_TO_WORD(srv.startAddressTI + i);
				event.value.ti := ti[i].value;
				event.qds.value := ti[i].qds.value;
				event.timeshtamp := tim;
				srv.setEvent(evt_type:= RLTNU.IECEventTypes.TI, event := event);
			END_IF 
		END_FOR
		FOR i := 0 TO IEC_COUNT_M_ME_TF_1-1 DO
			IF tf[i].value <> iecDB_tf[i].value OR tf[i].qds.value <> iecDB_tf[i].qds.value THEN
				tf[i].value := iecDB_tf[i].value;
				tf[i].qds.value := iecDB_tf[i].qds.value;
				
				RLTNU.SysTimeRtc.SysTimeRtcHighResGet(pTimestamp := tim);				
				event.addressObjectInformation := UDINT_TO_WORD(srv.startAddressTI + i);
				event.value.tf := tf[i].value;
				event.qds.value := tf[i].qds.value;
				event.timeshtamp := tim;
				srv.setEvent(evt_type:= RLTNU.IECEventTypes.TF, event := event);
			END_IF 
		END_FOR
	10:
		FOR i := 0 TO IEC_COUNT_M_SP_TB_1-1 DO
			IF ts[i].siq.value <> iecDB_ts[i].siq.value THEN
				ts[i].siq.value := iecDB_ts[i].siq.value;
				
				RLTNU.SysTimeRtc.SysTimeRtcHighResGet(pTimestamp := tim);				
				event.addressObjectInformation := UDINT_TO_WORD(srv.startAddressTS + i);
				IF ts[i].siq.value.0 THEN event.value.ts := 1; ELSE event.value.ts := 0; END_IF
				event.qds.value := ts[i].siq.value;
				event.timeshtamp := tim;
				srv.setEvent(evt_type:= RLTNU.IECEventTypes.TS, event := event);
			END_IF
		END_FOR
		FOR i := 0 TO IEC_COUNT_M_ME_TE_1-1 DO
			IF ti[i].value <> iecDB_te[i].value OR ti[i].qds.value <> iecDB_te[i].qds.value THEN
				ti[i].value := iecDB_te[i].value;
				ti[i].qds.value := iecDB_te[i].qds.value;
				
				RLTNU.SysTimeRtc.SysTimeRtcHighResGet(pTimestamp := tim);				
				event.addressObjectInformation := UDINT_TO_WORD(srv.startAddressTI + i);
				event.value.ti := ti[i].value;
				event.qds.value := ti[i].qds.value;
				event.timeshtamp := tim;
				srv.setEvent(evt_type:= RLTNU.IECEventTypes.TI, event := event);
			END_IF 
		END_FOR
		FOR i := 0 TO IEC_COUNT_M_ME_TF_1-1 DO
			IF tf[i].value <> iecDB_tf[i].value OR tf[i].qds.value <> iecDB_tf[i].qds.value THEN
				tf[i].value := iecDB_tf[i].value;
				tf[i].qds.value := iecDB_tf[i].qds.value;
				
				RLTNU.SysTimeRtc.SysTimeRtcHighResGet(pTimestamp := tim);				
				event.addressObjectInformation := UDINT_TO_WORD(srv.startAddressTF + i);
				event.value.tf := tf[i].value;
				event.qds.value := tf[i].qds.value;
				event.timeshtamp := tim;
				srv.setEvent(evt_type:= RLTNU.IECEventTypes.TF, event := event);
			END_IF 
		END_FOR
		state := 15;
	15:
		state := 20;
		srv();
		IF srv.error THEN
			state := 1000;
		END_IF
	20:
		state := 10;
		
		IF srv.getCommand(ADR(command)) THEN
			CASE(command.typeIdentifier) OF
				CMD_IDENT_C_SC_NA_1:
					IF InRange(command.addressObjectInformation, CMD_RANGE_C_SC_NA_1) THEN
						IF command.addressObjectInformation = ADRBASE_IEC_C_SC_NA_1 THEN
							options.last_group := (command.originator);
							// ПОКА ЧТО не делаем сохранение последнего центра, т.к. проще выдать команду "забрать управление".
							i := 0; WHILE i < COUNT_MAX_SERVERS DO
								IF station.originators[i] = options.last_group THEN
									EXIT;
								END_IF
								i := i + 1;
							END_WHILE
							IF i < COUNT_MAX_SERVERS THEN
								station.fail_center[i] := FALSE;
							END_IF
							srv.ackCommand(command, TRUE);
						ELSIF options.last_group = command.originator THEN
							iecDB_tu[command.addressObjectInformation-ADRBASE_IEC_C_SC_NA_1] := command.value.ts.0;
							iecDB_tu_act[command.addressObjectInformation-ADRBASE_IEC_C_SC_NA_1] := TRUE;
							srv.ackCommand(command, TRUE);
						ELSE
							i := 0; WHILE i < COUNT_MAX_SERVERS DO
								station.fail_control := TRUE;
								IF station.originators[i] = command.originator THEN
									station.fail_center[i] := TRUE;
								END_IF
								i := i + 1;
							END_WHILE
							srv.ackCommand(command, FALSE);
						END_IF
					ELSE
						srv.ackCommand(command, FALSE);
					END_IF
				
				CMD_IDENT_C_SE_NB_1:
					IF InRange(command.addressObjectInformation, CMD_RANGE_C_SE_NB_1) THEN
						IF options.last_group = command.originator THEN					
							srv.ackCommand(command, TRUE);
							iecDB_tri[command.addressObjectInformation-ADRBASE_IEC_C_SE_NB_1] := WORD_TO_UINT(command.value.ti);
							iecDB_tri_act[command.addressObjectInformation-ADRBASE_IEC_C_SE_NB_1] := TRUE;
						ELSE
							i := 0; WHILE i < COUNT_MAX_SERVERS DO
								station.fail_control := TRUE;
								IF station.originators[i] = command.originator THEN
									station.fail_center[i] := TRUE;
								END_IF
								i := i + 1;
							END_WHILE
							srv.ackCommand(command, FALSE);
						END_IF
					ELSE
						srv.ackCommand(command, FALSE);
					END_IF
				
				CMD_IDENT_C_SE_NC_1:
					IF InRange(command.addressObjectInformation, CMD_RANGE_C_SE_NC_1) THEN
						IF options.last_group = command.originator THEN					
							srv.ackCommand(command, TRUE);
							iecDB_trf[command.addressObjectInformation-ADRBASE_IEC_C_SE_NC_1] := command.value.tf;
							iecDB_trf_act[command.addressObjectInformation-ADRBASE_IEC_C_SE_NC_1] := TRUE;
						ELSE
							i := 0; WHILE i < COUNT_MAX_SERVERS DO
								station.fail_control := TRUE;
								IF station.originators[i] = command.originator THEN
									station.fail_center[i] := TRUE;
								END_IF
								i := i + 1;
							END_WHILE
							srv.ackCommand(command, FALSE);
						END_IF
					ELSE
						srv.ackCommand(command, FALSE);
					END_IF
				
				ELSE
					srv.ackCommand(command, FALSE);
			END_CASE
		END_IF		
		
	1000:
		srv.reset();
		state := 0;
END_CASE

METHOD PRIVATE InRange : BOOL
VAR_INPUT
	addr: WORD;
	typ: BYTE;
END_VAR
InRange := 0;
CASE(typ) OF
	CMD_RANGE_C_SC_NA_1:
	IF db.tu_count <> 0 THEN
		IF addr >= srv.startAddressTU AND addr < srv.startAddressTU + db.tu_count THEN
			InRange := 1;
		END_IF
	END_IF
	
	CMD_RANGE_C_SE_NB_1:
	IF db.tri_count <> 0 THEN
		IF addr >= srv.startAddressTRI AND addr < srv.startAddressTRI + db.tri_count THEN
			InRange := 1;
		END_IF
	END_IF
	
	CMD_RANGE_C_SE_NC_1:
	IF db.trf_count <> 0 THEN
		IF addr >= srv.startAddressTRF AND addr < srv.startAddressTRF + db.trf_count THEN
			InRange := 1;
		END_IF
	END_IF
	
END_CASE
END_METHOD

END_PROGRAM

// A1_01A/Application/Devices/TS
FUNCTION_BLOCK TS EXTENDS RLTM.DeviceTemplate
VAR_INPUT
END_VAR
VAR_OUTPUT
	tf: ARRAY[0..21] OF RLTNU.IEC_M_ME_NC;
END_VAR
VAR
	data_real: ARRAY[0..21] OF REAL;
	res: ARRAY[0..9] OF RLTM.RLTM_MODBUS_TRANSACTION_RESULT;
	i, j: UINT;
	c: ARRAY[0..15] OF UINT := [ 16#1, 16#2, 16#4, 16#8, 16#10, 16#20, 16#40, 16#80, 16#100, 16#200, 16#400, 16#800, 16#1000, 16#2000, 16#4000, 16#8000 ];
END_VAR

(*
Давление
Температура
Абсолютное давление
Коэффициент коррекции 
Коэффициент сжимаемости газа
Содержание азота
Содержание водорода
Содержание двуокиси углерода
Плость газа при нормальных условиях
Рабочий расход газа
Стандартный расход газа
Мощность
Теплотворная способность
Коэффициент плотности
Давление
Температура
Рабочий объём
Стандартный объём
Энергия
Рабочий расход прошлые сутки
Стандартный расход прошлые сутки
Рабочий расход прошлый месяц
Стандартный расход прошлый месяц
*)
FOR i := 0 TO 0 DO
	CASE res[i] OF
		RLTM.RLTM_TRANSACTION_RESULT_PROCESSING:
			;//nothing to do
		RLTM.RLTM_TRANSACTION_RESULT_SUCCESS:
			CASE i OF
				0:
					FOR j := 0 TO 23 DO
						tf[j].value := data_real[j];
						tf[j].qds.b.IV := 0;
					END_FOR
				
			END_CASE
	ELSE
		CASE i OF
				0:
					FOR j := 0 TO 23 DO
						tf[j].qds.b.IV := 1;
					END_FOR
		END_CASE
	END_CASE
END_FOR

METHOD Init: BOOL;
VAR_INPUT
END_VAR
VAR

END_VAR
SUPER^.Init();
transaction.typ := RLTM.RLTM_TRANSACTION_TYP_DATA;
transaction.mfc := 3;
transaction.offset := 0;
transaction.len := 46;
transaction.swap_byte := 1;
transaction.pData := ADR(data_real[0]);
transaction.pRes := ADR(res[0]);
transaction.timer.PT := T#1S;
SUPER^.AppendTransaction();

Init := 1;
END_METHOD

END_FUNCTION_BLOCK

// A1_01A/Application/Devices
PROGRAM Devices
VAR_INPUT
	enable: BOOL;
END_VAR
VAR
	state: INT := 0;
	i: UINT;
END_VAR

IF NOT enable THEN
	RETURN;
END_IF
// Виртуальные порты на Eth1 - начинаются со 100, на Eth2 - с 200
(* ================================================== *)

CASE state OF
	0:	// Инициализация виртуальных портов
		// ports param @ Init_Gen
		IF COUNT_PORT_ETH > 0 THEN
			DaemonIP.enable := TRUE;
		END_IF
		IF COUNT_PORT_SERIAL > 0 THEN
			DaemonSerial.enable := TRUE;
		END_IF
		state := 10;
		
	10:
		// Стартуем мастеров
		i := 0; WHILE i < COUNT_PORT_ETH DO
			modbus_ip[i].iif := DaemonIP.port_eth[i];	
			modbus_ip[i].activate := 1;
			modbus_ip[i].responseTimeout := T#1S;
			modbus_ip[i].Init(db_elements := 1);
			i := i + 1;
		END_WHILE
		i := 0; WHILE i < COUNT_PORT_SERIAL DO
			modbus_rs[i].iif := DaemonSerial.port_serial[i];	
			modbus_rs[i].activate := 1;
			modbus_rs[i].responseTimeout := T#1S;
			modbus_rs[i].Init(db_elements := 1);
			i := i + 1;
		END_WHILE
		
		// Инициализация устройств
		Init_Gen();
		state := 20;
		
		// Если для устройств задано кастомное значение каких-либо размерностей массивов из-за лишних резервов (тс, ти, команды...), 
		// нужно сообщить блоку количество переменных. Как правило, его можно взять из БД ВУ. Все параметры обязательны.
		// Пример (если задание параметров не сделано через скрипт в Devices.Init_Gen): ngk_ipkz_xn[0].SetCount(8, 3, 15, 5, 0, 4);

	20:
		// Вызов устройств
		i := 0; WHILE i < COUNT_PORT_ETH DO
			modbus_ip[i]();
			i := i + 1;
		END_WHILE
		i := 0; WHILE i < COUNT_PORT_SERIAL DO
			modbus_rs[i]();
			i := i + 1;
		END_WHILE
		
		Cyclic_Gen();
		
		Cyclic_DB();
END_CASE

METHOD Init_Gen
VAR_INPUT
END_VAR
    skp.node := 1;
    skp.pMaster := ADR(modbus_rs[0]);
    skp.Init();
    akp.node := 1;
    akp.pMaster := ADR(modbus_ip[0]);
    akp.Init();
    vopetm.node := 1;
    vopetm.pMaster := ADR(modbus_rs[1]);
    vopetm.Init();
    mercury.node := 1;
    mercury.pMaster := ADR(modbus_rs[1]);
    mercury.Init();
	(*
    ngk_ipkz_xn.node := 1;
    ngk_ipkz_xn.pMaster := ADR(modbus_rs[1]);
    ngk_ipkz_xn.Init();
	*)
    eris.node := 1;
    eris.pMaster := ADR(modbus_rs[1]);
    eris.Init();
    testGRS.node := 1;
    testGRS.pMaster := ADR(modbus_rs[1]);
    testGRS.Init();
    
    //ngk_ipkz_xn.SetCount(8, 9, 11, 5, 0, 4);
END_METHOD

METHOD Cyclic_Gen
VAR_INPUT
END_VAR
    skp();
    akp();
   (* vopetm();
    mercury();
    ngk_ipkz_xn();
    eris();
    testGRS();
*)
END_METHOD

METHOD Cyclic_DB
VAR_INPUT
END_VAR
VAR
	c_ts, c_te, c_tf, c_cmd, c_nb, c_nc: UDINT;
	i : UINT;
END_VAR
c_ts := ADRBASE_TS_DEVICE;
c_te := ADRBASE_TE_DEVICE;
c_tf := ADRBASE_TF_DEVICE;
c_cmd := ADRBASE_CMD_DEVICE;
c_nb := ADRBASE_NB_DEVICE;
c_nc := ADRBASE_NC_DEVICE;

{IF defined (variable: skp.ts)}
    i := 0; WHILE i < skp.count_ts DO
        iecDB_ts[c_ts + i] := skp.ts[i];
        i := i + 1;
    END_WHILE
    c_ts := c_ts + i;
{END_IF}
{IF defined (variable: skp.te)}
    i := 0; WHILE i < skp.count_te DO
        iecDB_te[c_te + i] := skp.te[i];
        i := i + 1;
    END_WHILE
    c_te := c_te + i;
{END_IF}
{IF defined (variable: skp.tf)}
    i := 0; WHILE i < skp.count_tf DO
        iecDB_tf[c_tf + i] := skp.tf[i];
        i := i + 1;
    END_WHILE
    c_tf := c_tf + i;
{END_IF}
{IF defined (variable: skp.cmd)}
    i := 0; WHILE i < skp.count_cmd DO
        IF iecDB_tu_act[c_cmd + i] THEN
            iecDB_tu_act[c_cmd + i] := FALSE;
            skp.cmd[i].run := TRUE;
            skp.cmd[i].value.spb := iecDB_tu[c_cmd + i];
        END_IF
        i := i + 1;
    END_WHILE
    c_cmd := c_cmd + i;
{END_IF}
{IF defined (variable: skp.nb)}
    i := 0; WHILE i < skp.count_nb DO
        IF iecDB_tri_act[c_nb + i] THEN
            iecDB_tri_act[c_nb + i] := FALSE;
            skp.nb[i].run := TRUE;
            skp.nb[i].value.spi := iecDB_tri[c_nb + i];
        END_IF
        i := i + 1;
    END_WHILE
    c_nb := c_nb + i;
{END_IF}
{IF defined (variable: skp.nc)}
    i := 0; WHILE i < skp.count_nc DO
        IF iecDB_trf_act[c_nc + i] THEN
            iecDB_trf_act[c_nc + i] := FALSE;
            skp.nc[i].run := TRUE;
            skp.nc[i].value.spr := iecDB_trf[c_nc + i];
        END_IF
        i := i + 1;
    END_WHILE
    c_nc := c_nc + i;
{END_IF}

{IF defined (variable: akp.ts)}
    i := 0; WHILE i < akp.count_ts DO
        iecDB_ts[c_ts + i] := akp.ts[i];
        i := i + 1;
    END_WHILE
    c_ts := c_ts + i;
{END_IF}
{IF defined (variable: akp.te)}
    i := 0; WHILE i < akp.count_te DO
        iecDB_te[c_te + i] := akp.te[i];
        i := i + 1;
    END_WHILE
    c_te := c_te + i;
{END_IF}
{IF defined (variable: akp.tf)}
    i := 0; WHILE i < akp.count_tf DO
        iecDB_tf[c_tf + i] := akp.tf[i];
        i := i + 1;
    END_WHILE
    c_tf := c_tf + i;
{END_IF}
{IF defined (variable: akp.cmd)}
    i := 0; WHILE i < akp.count_cmd DO
        IF iecDB_tu_act[c_cmd + i] THEN
            iecDB_tu_act[c_cmd + i] := FALSE;
            akp.cmd[i].run := TRUE;
            akp.cmd[i].value.spb := iecDB_tu[c_cmd + i];
        END_IF
        i := i + 1;
    END_WHILE
    c_cmd := c_cmd + i;
{END_IF}
{IF defined (variable: akp.nb)}
    i := 0; WHILE i < akp.count_nb DO
        IF iecDB_tri_act[c_nb + i] THEN
            iecDB_tri_act[c_nb + i] := FALSE;
            akp.nb[i].run := TRUE;
            akp.nb[i].value.spi := iecDB_tri[c_nb + i];
        END_IF
        i := i + 1;
    END_WHILE
    c_nb := c_nb + i;
{END_IF}
{IF defined (variable: akp.nc)}
    i := 0; WHILE i < akp.count_nc DO
        IF iecDB_trf_act[c_nc + i] THEN
            iecDB_trf_act[c_nc + i] := FALSE;
            akp.nc[i].run := TRUE;
            akp.nc[i].value.spr := iecDB_trf[c_nc + i];
        END_IF
        i := i + 1;
    END_WHILE
    c_nc := c_nc + i;
{END_IF}

{IF defined (variable: vopetm.ts)}
    i := 0; WHILE i < vopetm.count_ts DO
        iecDB_ts[c_ts + i] := vopetm.ts[i];
        i := i + 1;
    END_WHILE
    c_ts := c_ts + i;
{END_IF}
{IF defined (variable: vopetm.te)}
    i := 0; WHILE i < vopetm.count_te DO
        iecDB_te[c_te + i] := vopetm.te[i];
        i := i + 1;
    END_WHILE
    c_te := c_te + i;
{END_IF}
{IF defined (variable: vopetm.tf)}
    i := 0; WHILE i < vopetm.count_tf DO
        iecDB_tf[c_tf + i] := vopetm.tf[i];
        i := i + 1;
    END_WHILE
    c_tf := c_tf + i;
{END_IF}
{IF defined (variable: vopetm.cmd)}
    i := 0; WHILE i < vopetm.count_cmd DO
        IF iecDB_tu_act[c_cmd + i] THEN
            iecDB_tu_act[c_cmd + i] := FALSE;
            vopetm.cmd[i].run := TRUE;
            vopetm.cmd[i].value.spb := iecDB_tu[c_cmd + i];
        END_IF
        i := i + 1;
    END_WHILE
    c_cmd := c_cmd + i;
{END_IF}
{IF defined (variable: vopetm.nb)}
    i := 0; WHILE i < vopetm.count_nb DO
        IF iecDB_tri_act[c_nb + i] THEN
            iecDB_tri_act[c_nb + i] := FALSE;
            vopetm.nb[i].run := TRUE;
            vopetm.nb[i].value.spi := iecDB_tri[c_nb + i];
        END_IF
        i := i + 1;
    END_WHILE
    c_nb := c_nb + i;
{END_IF}
{IF defined (variable: vopetm.nc)}
    i := 0; WHILE i < vopetm.count_nc DO
        IF iecDB_trf_act[c_nc + i] THEN
            iecDB_trf_act[c_nc + i] := FALSE;
            vopetm.nc[i].run := TRUE;
            vopetm.nc[i].value.spr := iecDB_trf[c_nc + i];
        END_IF
        i := i + 1;
    END_WHILE
    c_nc := c_nc + i;
{END_IF}

{IF defined (variable: mercury.ts)}
    i := 0; WHILE i < mercury.count_ts DO
        iecDB_ts[c_ts + i] := mercury.ts[i];
        i := i + 1;
    END_WHILE
    c_ts := c_ts + i;
{END_IF}
{IF defined (variable: mercury.te)}
    i := 0; WHILE i < mercury.count_te DO
        iecDB_te[c_te + i] := mercury.te[i];
        i := i + 1;
    END_WHILE
    c_te := c_te + i;
{END_IF}
{IF defined (variable: mercury.tf)}
    i := 0; WHILE i < mercury.count_tf DO
        iecDB_tf[c_tf + i] := mercury.tf[i];
        i := i + 1;
    END_WHILE
    c_tf := c_tf + i;
{END_IF}
{IF defined (variable: mercury.cmd)}
    i := 0; WHILE i < mercury.count_cmd DO
        IF iecDB_tu_act[c_cmd + i] THEN
            iecDB_tu_act[c_cmd + i] := FALSE;
            mercury.cmd[i].run := TRUE;
            mercury.cmd[i].value.spb := iecDB_tu[c_cmd + i];
        END_IF
        i := i + 1;
    END_WHILE
    c_cmd := c_cmd + i;
{END_IF}
{IF defined (variable: mercury.nb)}
    i := 0; WHILE i < mercury.count_nb DO
        IF iecDB_tri_act[c_nb + i] THEN
            iecDB_tri_act[c_nb + i] := FALSE;
            mercury.nb[i].run := TRUE;
            mercury.nb[i].value.spi := iecDB_tri[c_nb + i];
        END_IF
        i := i + 1;
    END_WHILE
    c_nb := c_nb + i;
{END_IF}
{IF defined (variable: mercury.nc)}
    i := 0; WHILE i < mercury.count_nc DO
        IF iecDB_trf_act[c_nc + i] THEN
            iecDB_trf_act[c_nc + i] := FALSE;
            mercury.nc[i].run := TRUE;
            mercury.nc[i].value.spr := iecDB_trf[c_nc + i];
        END_IF
        i := i + 1;
    END_WHILE
    c_nc := c_nc + i;
{END_IF}

{IF defined (variable: ngk_ipkz_xn.ts)}
    i := 0; WHILE i < ngk_ipkz_xn.count_ts DO
        iecDB_ts[c_ts + i] := ngk_ipkz_xn.ts[i];
        i := i + 1;
    END_WHILE
    c_ts := c_ts + i;
{END_IF}
{IF defined (variable: ngk_ipkz_xn.te)}
    i := 0; WHILE i < ngk_ipkz_xn.count_te DO
        iecDB_te[c_te + i] := ngk_ipkz_xn.te[i];
        i := i + 1;
    END_WHILE
    c_te := c_te + i;
{END_IF}
{IF defined (variable: ngk_ipkz_xn.tf)}
    i := 0; WHILE i < ngk_ipkz_xn.count_tf DO
        iecDB_tf[c_tf + i] := ngk_ipkz_xn.tf[i];
        i := i + 1;
    END_WHILE
    c_tf := c_tf + i;
{END_IF}
{IF defined (variable: ngk_ipkz_xn.cmd)}
    i := 0; WHILE i < ngk_ipkz_xn.count_cmd DO
        IF iecDB_tu_act[c_cmd + i] THEN
            iecDB_tu_act[c_cmd + i] := FALSE;
            ngk_ipkz_xn.cmd[i].run := TRUE;
            ngk_ipkz_xn.cmd[i].value.spb := iecDB_tu[c_cmd + i];
        END_IF
        i := i + 1;
    END_WHILE
    c_cmd := c_cmd + i;
{END_IF}
{IF defined (variable: ngk_ipkz_xn.nb)}
    i := 0; WHILE i < ngk_ipkz_xn.count_nb DO
        IF iecDB_tri_act[c_nb + i] THEN
            iecDB_tri_act[c_nb + i] := FALSE;
            ngk_ipkz_xn.nb[i].run := TRUE;
            ngk_ipkz_xn.nb[i].value.spi := iecDB_tri[c_nb + i];
        END_IF
        i := i + 1;
    END_WHILE
    c_nb := c_nb + i;
{END_IF}
{IF defined (variable: ngk_ipkz_xn.nc)}
    i := 0; WHILE i < ngk_ipkz_xn.count_nc DO
        IF iecDB_trf_act[c_nc + i] THEN
            iecDB_trf_act[c_nc + i] := FALSE;
            ngk_ipkz_xn.nc[i].run := TRUE;
            ngk_ipkz_xn.nc[i].value.spr := iecDB_trf[c_nc + i];
        END_IF
        i := i + 1;
    END_WHILE
    c_nc := c_nc + i;
{END_IF}

{IF defined (variable: eris.ts)}
    i := 0; WHILE i < eris.count_ts DO
        iecDB_ts[c_ts + i] := eris.ts[i];
        i := i + 1;
    END_WHILE
    c_ts := c_ts + i;
{END_IF}
{IF defined (variable: eris.te)}
    i := 0; WHILE i < eris.count_te DO
        iecDB_te[c_te + i] := eris.te[i];
        i := i + 1;
    END_WHILE
    c_te := c_te + i;
{END_IF}
{IF defined (variable: eris.tf)}
    i := 0; WHILE i < eris.count_tf DO
        iecDB_tf[c_tf + i] := eris.tf[i];
        i := i + 1;
    END_WHILE
    c_tf := c_tf + i;
{END_IF}
{IF defined (variable: eris.cmd)}
    i := 0; WHILE i < eris.count_cmd DO
        IF iecDB_tu_act[c_cmd + i] THEN
            iecDB_tu_act[c_cmd + i] := FALSE;
            eris.cmd[i].run := TRUE;
            eris.cmd[i].value.spb := iecDB_tu[c_cmd + i];
        END_IF
        i := i + 1;
    END_WHILE
    c_cmd := c_cmd + i;
{END_IF}
{IF defined (variable: eris.nb)}
    i := 0; WHILE i < eris.count_nb DO
        IF iecDB_tri_act[c_nb + i] THEN
            iecDB_tri_act[c_nb + i] := FALSE;
            eris.nb[i].run := TRUE;
            eris.nb[i].value.spi := iecDB_tri[c_nb + i];
        END_IF
        i := i + 1;
    END_WHILE
    c_nb := c_nb + i;
{END_IF}
{IF defined (variable: eris.nc)}
    i := 0; WHILE i < eris.count_nc DO
        IF iecDB_trf_act[c_nc + i] THEN
            iecDB_trf_act[c_nc + i] := FALSE;
            eris.nc[i].run := TRUE;
            eris.nc[i].value.spr := iecDB_trf[c_nc + i];
        END_IF
        i := i + 1;
    END_WHILE
    c_nc := c_nc + i;
{END_IF}

{IF defined (variable: testGRS.ts)}
    i := 0; WHILE i < testGRS.count_ts DO
        iecDB_ts[c_ts + i] := testGRS.ts[i];
        i := i + 1;
    END_WHILE
    c_ts := c_ts + i;
{END_IF}
{IF defined (variable: testGRS.te)}
    i := 0; WHILE i < testGRS.count_te DO
        iecDB_te[c_te + i] := testGRS.te[i];
        i := i + 1;
    END_WHILE
    c_te := c_te + i;
{END_IF}
{IF defined (variable: testGRS.tf)}
    i := 0; WHILE i < testGRS.count_tf DO
        iecDB_tf[c_tf + i] := testGRS.tf[i];
        i := i + 1;
    END_WHILE
    c_tf := c_tf + i;
{END_IF}
{IF defined (variable: testGRS.cmd)}
    i := 0; WHILE i < testGRS.count_cmd DO
        IF iecDB_tu_act[c_cmd + i] THEN
            iecDB_tu_act[c_cmd + i] := FALSE;
            testGRS.cmd[i].run := TRUE;
            testGRS.cmd[i].value.spb := iecDB_tu[c_cmd + i];
        END_IF
        i := i + 1;
    END_WHILE
    c_cmd := c_cmd + i;
{END_IF}
{IF defined (variable: testGRS.nb)}
    i := 0; WHILE i < testGRS.count_nb DO
        IF iecDB_tri_act[c_nb + i] THEN
            iecDB_tri_act[c_nb + i] := FALSE;
            testGRS.nb[i].run := TRUE;
            testGRS.nb[i].value.spi := iecDB_tri[c_nb + i];
        END_IF
        i := i + 1;
    END_WHILE
    c_nb := c_nb + i;
{END_IF}
{IF defined (variable: testGRS.nc)}
    i := 0; WHILE i < testGRS.count_nc DO
        IF iecDB_trf_act[c_nc + i] THEN
            iecDB_trf_act[c_nc + i] := FALSE;
            testGRS.nc[i].run := TRUE;
            testGRS.nc[i].value.spr := iecDB_trf[c_nc + i];
        END_IF
        i := i + 1;
    END_WHILE
    c_nc := c_nc + i;
{END_IF}
END_METHOD

END_PROGRAM

// A1_01A/Application/DaemonIP
PROGRAM DaemonIP
VAR_INPUT
	enable: BOOL;
	port_cfg_eth: ARRAY[0.._S_COUNT_PORT_ETH] OF RLTM.IP_CONFIG;
END_VAR
VAR
	port_eth: ARRAY[0.._S_COUNT_PORT_ETH] OF RLTM.CAA_IP;
	port_cyclic: ARRAY[0.._S_COUNT_PORT_ETH] OF BOOL;
	i: UINT;
	step: UINT;
END_VAR

IF NOT enable THEN
	RETURN;
END_IF

i := 0; WHILE i < COUNT_PORT_ETH DO
	IF NOT port_cyclic[i] THEN
		// инициализация порта
		IF port_cfg_eth[i].enable THEN
			port_eth[i].Start(pCfg := ADR(port_cfg_eth[i]));
		END_IF
		port_cyclic[i] := TRUE;
	ELSE
		// вызов циклической процедуры с частотой большей, чем у основной задачи
		port_cyclic[i] := port_eth[i].Cyclic();
	END_IF
	i := i + 1;
END_WHILE

END_PROGRAM

// A1_01A/Application/DaemonSerial
PROGRAM DaemonSerial
VAR_INPUT
	enable: BOOL;
	port_cfg_serial: ARRAY[0.._S_COUNT_PORT_SERIAL] OF RLTM.SERIAL_CONFIG;
END_VAR
VAR
	port_serial: ARRAY[0.._S_COUNT_PORT_SERIAL] OF RLTM.CAA_SERIAL;
	port_cyclic: ARRAY[0.._S_COUNT_PORT_SERIAL] OF BOOL;
	i: UINT;
	step: UINT;
END_VAR

IF NOT enable THEN
	RETURN;
END_IF

i := 0; WHILE i < COUNT_PORT_SERIAL DO
	IF NOT port_cyclic[i] THEN
		// инициализация порта
		IF port_cfg_serial[i].enable THEN
			port_serial[i].Start(pCfg := ADR(port_cfg_serial[i]));
		END_IF
		port_cyclic[i] := TRUE;
	ELSE
		// вызов циклической процедуры с частотой большей, чем у основной задачи
		port_cyclic[i] := port_serial[i].Cyclic();
	END_IF
	i := i + 1;
END_WHILE

END_PROGRAM

// A1_01A/Application/Devices/SKP
FUNCTION_BLOCK SKP EXTENDS RLTM.DeviceTemplate
VAR_INPUT
	cmd: ARRAY[0..54] OF RLTM.RLTM_MODBUS_CMD;
	//nc: ARRAY[0..3] OF RLTM.RLTM_MODBUS_CMD;
END_VAR
VAR_OUTPUT
	ts: ARRAY[0..110] OF RLTNU.IEC_M_SP_NA;
	te: ARRAY[0..31] OF RLTNU.IEC_M_ME_NB;
	//tf: ARRAY[0..26] OF RLTNU.IEC_M_ME_NC;
END_VAR
VAR
	//sp_cmd: ARRAY[0..4] OF BOOL;
	//sp0: ARRAY[0..4] OF INT;
	data_int: ARRAY[0..32] OF INT;
	res: ARRAY[0..9] OF RLTM.RLTM_MODBUS_TRANSACTION_RESULT;
	i, j: UINT;
	u: UDINT;
END_VAR

FOR i := 0 TO 1 DO
	CASE res[i] OF
		RLTM.RLTM_TRANSACTION_RESULT_PROCESSING:
			;//nothing to do
		RLTM.RLTM_TRANSACTION_RESULT_SUCCESS:
			CASE i OF
				0:
					FOR j := 0 TO 110 DO
						ts[j].siq.b.SPI := p_bool[j];
						ts[j].siq.b.IV := 0;
					END_FOR
					
				1:
					FOR j := 0 TO 31 DO
						te[j].value := p_uint[j];
						te[j].qds.b.IV := 0;
					END_FOR
					
			END_CASE
			res[i] := RLTM.RLTM_TRANSACTION_RESULT_PROCESSING;
		ELSE
			CASE i OF
				0:
					FOR j := 0 TO 110 DO
						ts[j].siq.b.IV := 1;
					END_FOR
				1:
					FOR j := 0 TO 32 DO
						te[j].qds.b.IV := 1;
					END_FOR
			END_CASE
		
		
	END_CASE
END_FOR

METHOD PUBLIC Init : BOOL
VAR_INPUT
END_VAR
VAR
	i:UINT;
END_VAR
SUPER^.Init();

(*	0x01 - 0x2C	*)
transaction.typ := RLTM.RLTM_TRANSACTION_TYP_DATA;
transaction.mfc := 2;
transaction.offset := 1024;
transaction.len := 110;
transaction.swap_byte := 1;
transaction.pData := ADR(buf[0]);
transaction.pRes := ADR(res[0]);
transaction.timer.PT := T#1S;
SUPER^.AppendTransaction();

(*	0x01 - 0x08	*)
transaction.typ := RLTM.RLTM_TRANSACTION_TYP_DATA;
transaction.mfc := 3;
transaction.offset := 2048;
transaction.len := 32;
transaction.swap_byte := 1;
transaction.pData := ADR(buf[0]);
transaction.pRes := ADR(res[1]);
transaction.timer.PT := T#1S;
SUPER^.AppendTransaction();

(*
FOR i := 0 TO 54 DO
	//0х0081  Дистанционное отключение и включение модулей силовых
	transaction.typ := RLTM.RLTM_TRANSACTION_TYP_CMD;
	transaction.mfc := 5;
	transaction.offset := 3072+i;
	transaction.len := 1;
	transaction.swap_byte := 0;
	transaction.pCmd := ADR(cmd[i].run);
	transaction.pData := ADR(cmd[i].value.spb);
	transaction.pRes := ADR(res[2]);
	transaction.timer.PT := T#1S;
	SUPER^.AppendTransaction();
END_FOR
*)
Init := 1;
END_METHOD

METHOD PUBLIC FB_init : BOOL
VAR_INPUT
	bInitRetains : BOOL; // if TRUE, the retain variables are initialized (warm start / cold start)
	bInCopyCode : BOOL;  // if TRUE, the instance afterwards gets moved into the copy code (online change)
END_VAR
// Определение размерностей (нужно во всех устройствах)
{IF defined (variable: ts)}
    count_ts := SIZEOF(ts)/SIZEOF(ts[0]);
{END_IF}
{IF defined (variable: te)}
    count_te := SIZEOF(te)/SIZEOF(te[0]);
{END_IF}
{IF defined (variable: tf)}
    count_tf := sizeof(tf)/sizeof(tf[0]);
{END_IF}
{IF defined (variable: cmd)}
    count_cmd := SIZEOF(cmd)/SIZEOF(cmd[0]);
{END_IF}
{IF defined (variable: nb)}
    count_nb := SIZEOF(nb)/SIZEOF(nb[0]);
{END_IF}
{IF defined (variable: nc)}
    count_nc := SIZEOF(nc)/SIZEOF(nc[0]);
{END_IF}
END_METHOD

METHOD SetCount
VAR_INPUT
	new_ts: UINT := 0;
	new_te: UINT := 0;
	new_tf: UINT := 0;
	new_cmd: UINT := 0;
	new_nb: UINT := 0;
	new_nc: UINT := 0;
END_VAR
	count_ts := new_ts;
	count_te := new_te;
	count_tf := new_tf;
	count_cmd := new_cmd;
	count_nb := new_nb;
	count_nc := new_nc;
END_METHOD

END_FUNCTION_BLOCK

// A1_01A/Application/Devices/AKP
FUNCTION_BLOCK AKP EXTENDS RLTM.DeviceTemplate
VAR_INPUT
	cmd: ARRAY[0..12] OF RLTM.RLTM_MODBUS_CMD;
	//nc: ARRAY[0..3] OF RLTM.RLTM_MODBUS_CMD;
END_VAR
VAR_OUTPUT
	ts: ARRAY[0..39] OF RLTNU.IEC_M_SP_NA;
	te: ARRAY[0..21] OF RLTNU.IEC_M_ME_NB;
	tf: ARRAY[0..15] OF RLTNU.IEC_M_ME_NC;
END_VAR
VAR
	//sp_cmd: ARRAY[0..4] OF BOOL;
	//sp0: ARRAY[0..4] OF INT;
	data_int: ARRAY[0..32] OF INT;
	res: ARRAY[0..9] OF RLTM.RLTM_MODBUS_TRANSACTION_RESULT;
	i, j: UINT;
	u: UDINT;
END_VAR

FOR i := 0 TO 1 DO
	CASE res[i] OF
		RLTM.RLTM_TRANSACTION_RESULT_PROCESSING:
			;//nothing to do
		RLTM.RLTM_TRANSACTION_RESULT_SUCCESS:
			CASE i OF
				0:
					FOR j := 0 TO 39 DO
						ts[j].siq.b.SPI := p_bool[j];
						ts[j].siq.b.IV := 0;
					END_FOR
					
				1:
					FOR j := 0 TO 21 DO
						te[j].value := p_uint[j];
						te[j].qds.b.IV := 0;
					END_FOR
					
				2:
					FOR j := 0 TO 15 DO
						tf[j].value := p_real[j];
						tf[j].qds.b.IV := 0;
					END_FOR	
			END_CASE
			res[i] := RLTM.RLTM_TRANSACTION_RESULT_PROCESSING;
		ELSE
			CASE i OF
				0:
					FOR j := 0 TO 39 DO
						ts[j].siq.b.IV := 1;
					END_FOR
				1:
					FOR j := 0 TO 21 DO
						te[j].qds.b.IV := 1;
					END_FOR
				2:
					FOR j := 0 TO 15 DO
						te[j].qds.b.IV := 1;
					END_FOR
				
			END_CASE
		
		
	END_CASE
END_FOR

METHOD PUBLIC Init : BOOL
VAR_INPUT
END_VAR
VAR
	i:UINT;
END_VAR
SUPER^.Init();

(*	0x01 - 0x2C	*)
transaction.typ := RLTM.RLTM_TRANSACTION_TYP_DATA;
transaction.mfc := 2;
transaction.offset := 1000;
transaction.len := 40;
transaction.swap_byte := 1;
transaction.pData := ADR(buf[0]);
transaction.pRes := ADR(res[0]);
transaction.timer.PT := T#1S;
SUPER^.AppendTransaction();

(*	0x01 - 0x08	*)
transaction.typ := RLTM.RLTM_TRANSACTION_TYP_DATA;
transaction.mfc := 3;
transaction.offset := 2000;
transaction.len := 22;
transaction.swap_byte := 1;
transaction.pData := ADR(buf[0]);
transaction.pRes := ADR(res[1]);
transaction.timer.PT := T#1S;
SUPER^.AppendTransaction();
(*
(*	0x01 - 0x08	*)
transaction.typ := RLTM.RLTM_TRANSACTION_TYP_DATA;
transaction.mfc := 3;
transaction.offset := 4000;
transaction.len := 16;
transaction.swap_byte := 1;
transaction.pData := ADR(buf[0]);
transaction.pRes := ADR(res[1]);
transaction.timer.PT := T#1S;
SUPER^.AppendTransaction();


FOR i := 0 TO 54 DO
	//0х0081  Дистанционное отключение и включение модулей силовых
	transaction.typ := RLTM.RLTM_TRANSACTION_TYP_CMD;
	transaction.mfc := 5;
	transaction.offset := 3072+i;
	transaction.len := 1;
	transaction.swap_byte := 0;
	transaction.pCmd := ADR(cmd[i].run);
	transaction.pData := ADR(cmd[i].value.spb);
	transaction.pRes := ADR(res[2]);
	transaction.timer.PT := T#1S;
	SUPER^.AppendTransaction();
END_FOR

*)



Init := 1;
END_METHOD

METHOD PUBLIC FB_init : BOOL
VAR_INPUT
	bInitRetains : BOOL; // if TRUE, the retain variables are initialized (warm start / cold start)
	bInCopyCode : BOOL;  // if TRUE, the instance afterwards gets moved into the copy code (online change)
END_VAR
// Определение размерностей (нужно во всех устройствах)
{IF defined (variable: ts)}
    count_ts := SIZEOF(ts)/SIZEOF(ts[0]);
{END_IF}
{IF defined (variable: te)}
    count_te := SIZEOF(te)/SIZEOF(te[0]);
{END_IF}
{IF defined (variable: tf)}
    count_tf := sizeof(tf)/sizeof(tf[0]);
{END_IF}
{IF defined (variable: cmd)}
    count_cmd := SIZEOF(cmd)/SIZEOF(cmd[0]);
{END_IF}
{IF defined (variable: nb)}
    count_nb := SIZEOF(nb)/SIZEOF(nb[0]);
{END_IF}
{IF defined (variable: nc)}
    count_nc := SIZEOF(nc)/SIZEOF(nc[0]);
{END_IF}
END_METHOD

METHOD SetCount
VAR_INPUT
	new_ts: UINT := 0;
	new_te: UINT := 0;
	new_tf: UINT := 0;
	new_cmd: UINT := 0;
	new_nb: UINT := 0;
	new_nc: UINT := 0;
END_VAR
	count_ts := new_ts;
	count_te := new_te;
	count_tf := new_tf;
	count_cmd := new_cmd;
	count_nb := new_nb;
	count_nc := new_nc;
END_METHOD

END_FUNCTION_BLOCK

// A1_01A/Application/Devices/Mercury
FUNCTION_BLOCK Mercury EXTENDS RLTM.DeviceTemplate
VAR_INPUT
END_VAR
VAR_OUTPUT
	tf: ARRAY[0..21] OF RLTNU.IEC_M_ME_NC;
END_VAR
VAR
	data_real: ARRAY[0..21] OF REAL;
	res: ARRAY[0..9] OF RLTM.RLTM_MODBUS_TRANSACTION_RESULT;
	i, j: UINT;
	c: ARRAY[0..15] OF UINT := [ 16#1, 16#2, 16#4, 16#8, 16#10, 16#20, 16#40, 16#80, 16#100, 16#200, 16#400, 16#800, 16#1000, 16#2000, 16#4000, 16#8000 ];
END_VAR

(*
Мгновенная активная мощность по фазе 1
Мгновенная активная мощность по фазе 2
Мгновенная активная мощность по фазе 3
Напряжение по фазе 1
Напряжение по фазе 2
Напряжение по фазе 3
Ток по фазе 1
Ток по фазе 2
Ток по фазе 3
Суммарная активная мощность от сброса
Суммарная активная мощность до сброса
Суммарная реактивная мощность от сброса
Суммарная реактивная мощность до сброса
Активная мощность от сброса за текущие сутки
Активная мощность до сброса за текущие сутки
Реактивная мощность от сброса за текущие сутки
Реактивная мощность до сброса за текущие сутки
Активная мощность от сброса за предыдущие сутки
Активная мощность до сброса за предыдущие сутки
Реактивная мощность от сброса за предыдущие сутки
Реактивная мощность до сброса за предыдущие сутки
*)
FOR i := 0 TO 0 DO
	CASE res[i] OF
		RLTM.RLTM_TRANSACTION_RESULT_PROCESSING:
			;//nothing to do
		RLTM.RLTM_TRANSACTION_RESULT_SUCCESS:
			CASE i OF
				0:
					FOR j := 0 TO 21 DO
						tf[j].value := data_real[j];
						tf[j].qds.b.IV := 0;
					END_FOR
				
			END_CASE
	ELSE
		CASE i OF
				0:
					FOR j := 0 TO 21 DO
						tf[j].qds.b.IV := 1;
					END_FOR
		END_CASE
	END_CASE
END_FOR

METHOD Init: BOOL;
VAR_INPUT
END_VAR
VAR

END_VAR
SUPER^.Init();
transaction.typ := RLTM.RLTM_TRANSACTION_TYP_DATA;
transaction.mfc := 3;
transaction.offset := 0;
transaction.len := 42;
transaction.swap_byte := 1;
transaction.pData := ADR(data_real[0]);
transaction.pRes := ADR(res[0]);
transaction.timer.PT := T#1S;
SUPER^.AppendTransaction();

Init := 1;
END_METHOD

END_FUNCTION_BLOCK

// A1_01A/Application/IP2RS_PRG
PROGRAM IP2RS_PRG
VAR CONSTANT

	client_conf : ARRAY [0..3] OF ClientCfg := [
				(client_address := '172.16.26.2', server_port := 2405, rs_port := 1, route_address := '127.0.0.1', route_port := 2405),
				(client_address := '172.16.26.3', server_port := 2405, rs_port := 1, route_address := '127.0.0.1', route_port := 2405),
				(client_address := '172.16.26.13', server_port := 2405, rs_port := 1, route_address := '127.0.0.1', route_port := 2405),
				(client_address := '', server_port := 0, rs_port := 0, route_address := '', route_port := 0)		// пустая строка должна быть в конце массива
	];
	
	serial_conf : ARRAY [0..1] OF SerialCfg := [
				(number := 1, baudrate := 9600, parity := COM_Parity.SYS_NOPARITY, stopbits := COM_StopBits.SYS_ONESTOPBIT, timeout := TIME_TO_UDINT(T#100MS), frame_size := 250, mode := SerialConst.HALF_SLAVE),
				(number := 0, baudrate := 0, parity := 0, stopbits := 0, timeout := 0, frame_size := 0, mode := 0)		// пустая строка должна быть в конце массива
	];
	
END_VAR
VAR
	buffers		: Exchange_Buffer;
	ports		: Serial_group;
	clients		: Client_group;

	bu, po, cl		:BOOL;
	first : BOOL := TRUE;
END_VAR

IF first THEN
	bu := buffers.Init(clientsCfg := ADR(client_conf), portsCfg := ADR(serial_conf));
	po := ports.Init(portsCfg := ADR(serial_conf), ip2rs_buffer := ADR(buffers));
	cl := clients.Init(clientsCfg := ADR(client_conf), ip2rs_buffer := ADR(buffers));
	first := FALSE;
END_IF

buffers();
ports();
clients();

END_PROGRAM

// Exchange/Exchange_Buffer
FUNCTION_BLOCK Exchange_Buffer
VAR_INPUT
END_VAR
VAR_OUTPUT
END_VAR
VAR
	from_ip			: POINTER TO IP_Buffer;
	from_rs			: POINTER TO IP_Buffer;
	size			: UINT;
END_VAR

METHOD AddRSMessage : BOOL
VAR_INPUT
	rs_port			: UINT;
	data			: POINTER TO BYTE;
	length			: UINT;
END_VAR
VAR
	i, pos			: UINT;
	msg				: POINTER TO IP_Message;
	data_length		: UINT;
	temp			: UDINT;
END_VAR

AddRSMessage := FALSE;

IF (from_rs = 0) OR (data = 0) OR (length < SIZEOF(msg^.ip_port) + SIZEOF(msg^.address) + SIZEOF(msg^.state)) 
				OR (length > SIZEOF(msg^.ip_port) + SIZEOF(msg^.address) + SIZEOF(msg^.state) + MSG_SIZE) THEN
		RETURN;
END_IF;

data_length := length - SIZEOF(msg^.ip_port) - SIZEOF(msg^.address) - SIZEOF(msg^.state);
			
FOR i := 0 TO THIS^.size - 1 DO	
	IF (from_rs[i].rs_port = rs_port) AND (from_rs[i].size <> 0) THEN
		msg := ADR(from_rs[i].messages[from_rs[i].end]);				
		IF from_rs[i].qnt < from_rs[i].size THEN				
			from_rs[i].qnt := from_rs[i].qnt + 1;
		ELSE
			from_rs[i].begin := (from_rs[i].begin + 1) MOD from_rs[i].size;				
		END_IF
		from_rs[i].end := (from_rs[i].end + 1) MOD from_rs[i].size;
		
		SysMemSet(msg, 0, SIZEOF(IP_Message));
		pos := 0;
		SysMemCpy(ADR(msg^.ip_port), ADR(data[pos]), SIZEOF(msg^.ip_port));
		pos := pos + SIZEOF(msg^.ip_port);		
		SysMemCpy(ADR(temp), ADR(data[pos]), SIZEOF(msg^.address));
		msg^.address := temp;
		pos := pos + SIZEOF(msg^.address);
		SysMemCpy(ADR(msg^.state), ADR(data[pos]), SIZEOF(msg^.state));
		pos := pos + SIZEOF(msg^.state);
		SysMemCpy(ADR(msg^.data[0]), ADR(data[pos]), data_length);
		msg^.length := data_length;
		
		AddRSMessage := TRUE;
		RETURN;
	END_IF
END_FOR
END_METHOD

METHOD fb_init : BOOL
VAR_INPUT
	bInitRetains : BOOL; // if TRUE, the retain variables are initialized (warm start / cold start)
	bInCopyCode : BOOL;  // if TRUE, the instance afterwards gets moved into the copy code (online change)

//	clientsCfg	: POINTER TO ClientCfg;
//	portsCfg	: POINTER TO SerialCfg;
END_VAR
VAR
	i, j		: UINT;
	result		: RTS_IEC_RESULT;
	msg_qnt		: UINT;
	name		: string;
END_VAR
(*
from_ip := 0;
from_rs := 0;
size := 0;

IF (clientsCfg = 0) OR (portsCfg = 0) THEN
	fb_init := FALSE;
	RETURN;
END_IF

i := 0;
WHILE (portsCfg[i].number > 0) DO
	i := i+1;
END_WHILE
IF i = 0 THEN
	fb_init := FALSE;
	RETURN;
END_IF

size := i;
name := UDINT_TO_STRING(ADR(from_ip));
from_ip := SysMemAllocData(name, size*SIZEOF(IP_Buffer), ADR(result));
name := UDINT_TO_STRING(ADR(from_rs));
from_rs := SysMemAllocData(name, size*SIZEOF(IP_Buffer), ADR(result));
IF (from_ip = 0) OR (from_rs = 0) THEN
	fb_init := FALSE;
	fb_exit(FALSE);
	RETURN;
END_IF
SysMemSet(from_ip, 0, size*SIZEOF(IP_Buffer));
SysMemSet(from_rs, 0, size*SIZEOF(IP_Buffer));

FOR i := 0 TO size - 1 DO	
	j := 0;
	msg_qnt := 0;
	WHILE (LEN(clientsCfg[j].client_address) > 0) DO		
		IF (clientsCfg[j].rs_port = portsCfg[i].number) THEN
			msg_qnt := msg_qnt +1;
		END_IF
		j := j+1;
	END_WHILE
	IF (msg_qnt <> 0) THEN		
		from_ip[i].size := msg_qnt*2;
		name := UDINT_TO_STRING(ADR(from_ip[i]));
		from_ip[i].messages := SysMemAllocData(name, from_ip[i].size*SIZEOF(IP_Message), ADR(result));
		from_rs[i].size := msg_qnt*4;
		name := UDINT_TO_STRING(ADR(from_rs[i]));
		from_rs[i].messages := SysMemAllocData(name, from_rs[i].size*SIZEOF(IP_Message), ADR(result));
		IF (from_ip[i].messages = 0) OR (from_rs[i].messages = 0) THEN
			fb_init := FALSE;
			fb_exit(FALSE);
			RETURN;
		END_IF
		SysMemSet(from_ip[i].messages, 0, from_ip[i].size*SIZEOF(IP_Message));
		SysMemSet(from_rs[i].messages, 0, from_rs[i].size*SIZEOF(IP_Message));
		from_ip[i].rs_port := portsCfg[i].number;
		from_rs[i].rs_port := portsCfg[i].number;
	END_IF	
END_FOR

fb_init := TRUE;
*)
END_METHOD

METHOD GetMessageForRS : BOOL
VAR_INPUT
	rs_port			: UINT;
	data			: POINTER TO BYTE;
	size			: UINT;
	length			: POINTER TO UINT;
END_VAR
VAR
	i, pos			: UINT;
	msg				: POINTER TO IP_Message;
	msg_length		: UINT;
	temp			: UDINT;
END_VAR

GetMessageForRS := FALSE;

IF (from_ip = 0) OR (data = 0) OR (length = 0) THEN
	RETURN;
END_IF

FOR i := 0 TO THIS^.size - 1 DO	
	IF (from_ip[i].rs_port = rs_port) AND (from_ip[i].size <> 0) THEN			
		WHILE (from_ip[i].qnt <> 0) DO			
			msg := ADR(from_ip[i].messages[from_ip[i].begin]);
			from_ip[i].begin := (from_ip[i].begin + 1) MOD from_ip[i].size;
			from_ip[i].qnt := from_ip[i].qnt - 1;
			
			msg_length := SIZEOF(msg^.ip_port) + SIZEOF(msg^.address) + SIZEOF(msg^.state) + msg^.length;			
			IF (msg_length > size) THEN CONTINUE; END_IF;
			
			pos := 0;
			SysMemCpy(ADR(data[pos]), ADR(msg^.ip_port), SIZEOF(msg^.ip_port));
			pos := pos + SIZEOF(msg^.ip_port);
			temp := msg^.address;
			SysMemCpy(ADR(data[pos]), ADR(temp), SIZEOF(msg^.address));
			pos := pos + SIZEOF(msg^.address);
			SysMemCpy(ADR(data[pos]), ADR(msg^.state), SIZEOF(msg^.state));
			pos := pos + SIZEOF(msg^.state);
			SysMemCpy(ADR(data[pos]), ADR(msg^.data[0]), msg^.length);
			length^ := msg_length;
			
			GetMessageForRS := TRUE;
			RETURN;
		END_WHILE
	END_IF
END_FOR
END_METHOD

METHOD ClearByClient
VAR_INPUT
	ip_port			: UINT;
	address			: UDINT;
	rs_port			: UINT;	
END_VAR
VAR
	i				: UINT;
	local_begin		: UINT;
	local_qnt		: UINT;
	msg				: POINTER TO IP_Message;
END_VAR
IF (from_ip = 0) OR (from_rs = 0) THEN
	RETURN;
END_IF

FOR i := 0 TO THIS^.size - 1 DO	
	IF (from_ip[i].rs_port = rs_port) AND (from_ip[i].size <> 0) THEN
		local_begin := from_ip[i].begin;
		local_qnt := from_ip[i].qnt;
		WHILE (local_qnt <> 0) DO
			msg := ADR(from_ip[i].messages[local_begin]);			
			IF (msg^.ip_port = ip_port) AND (msg^.address = address) THEN
				DeleteMessage(ADR(from_ip[i]), local_begin);
			END_IF			
			local_begin := (local_begin + 1) MOD from_ip[i].size;
			local_qnt := local_qnt - 1;
		END_WHILE
	END_IF
	IF (from_rs[i].rs_port = rs_port) AND (from_rs[i].size <> 0) THEN
		local_begin := from_rs[i].begin;
		local_qnt := from_rs[i].qnt;
		WHILE (local_qnt <> 0) DO
			msg := ADR(from_rs[i].messages[local_begin]);			
			IF (msg^.ip_port = ip_port) AND (msg^.address = address) THEN
				DeleteMessage(ADR(from_rs[i]), local_begin);
			END_IF			
			local_begin := (local_begin + 1) MOD from_rs[i].size;
			local_qnt := local_qnt - 1;
		END_WHILE
	END_IF
END_FOR
END_METHOD

METHOD AddIPMessage : BOOL
VAR_INPUT
	ip_port			: UINT;
	address			: UDINT;
	rs_port			: UINT;
	state			: UINT;
	data			: POINTER TO BYTE;
	length			: UINT;
END_VAR
VAR
	i				: UINT;
	msg				: POINTER TO IP_Message;
END_VAR

AddIPMessage := FALSE;

IF (from_ip = 0) OR (data = 0) OR (length > MSG_SIZE) THEN
	RETURN;
END_IF;

FOR i := 0 TO THIS^.size - 1 DO	
	IF (from_ip[i].rs_port = rs_port) AND (from_ip[i].size <> 0) THEN
		msg := ADR(from_ip[i].messages[from_ip[i].end]);				
		IF from_ip[i].qnt < from_ip[i].size THEN				
			from_ip[i].qnt := from_ip[i].qnt + 1;
		ELSE
			from_ip[i].begin := (from_ip[i].begin + 1) MOD from_ip[i].size;				
		END_IF
		from_ip[i].end := (from_ip[i].end + 1) MOD from_ip[i].size;
		
		SysMemSet(msg, 0, SIZEOF(IP_Message));
		msg^.ip_port := ip_port;		
		msg^.address := address;
		msg^.state := state;
		SysMemCpy(ADR(msg^.data[0]), data, length);
		msg^.length := length;		
		AddIPMessage := TRUE;
		RETURN;
	END_IF
END_FOR
END_METHOD

METHOD CheckIPMessage : UINT
VAR_INPUT
	ip_port			: UINT;
	address			: UDINT;
	rs_port			: UINT;
END_VAR
VAR
	i				: UINT;
	local_begin		: UINT;
	local_qnt		: UINT;
	msg				: POINTER TO IP_Message;
END_VAR

CheckIPMessage := 0;

IF (from_ip = 0) THEN
	RETURN;
END_IF;

FOR i := 0 TO THIS^.size - 1 DO	
	IF (from_ip[i].rs_port = rs_port) AND (from_ip[i].size <> 0) THEN
		local_begin := from_ip[i].begin;
		local_qnt := from_ip[i].qnt;
		WHILE (local_qnt <> 0) DO
			msg := ADR(from_ip[i].messages[local_begin]);			
			IF (msg^.ip_port = ip_port) AND (msg^.address = address) THEN
				CheckIPMessage := CheckIPMessage + 1;
			END_IF			
			local_begin := (local_begin + 1) MOD from_ip[i].size;
			local_qnt := local_qnt - 1;
		END_WHILE
	END_IF
END_FOR
END_METHOD

METHOD Init : BOOL
VAR_INPUT
	clientsCfg	: POINTER TO ClientCfg;
	portsCfg	: POINTER TO SerialCfg;
END_VAR
VAR
	i, j		: UINT;
	result		: RTS_IEC_RESULT;
	msg_qnt		: UINT;
	name		: string;
END_VAR

from_ip := 0;
from_rs := 0;
size := 0;

IF (clientsCfg = 0) OR (portsCfg = 0) THEN
	Init := FALSE;
	RETURN;
END_IF

i := 0;
WHILE (portsCfg[i].number > 0) DO
	i := i+1;
END_WHILE
IF i = 0 THEN
	Init := FALSE;
	RETURN;
END_IF

size := i;
name := UDINT_TO_STRING(ADR(from_ip));
from_ip := SysMemAllocData(name, size*SIZEOF(IP_Buffer), ADR(result));
name := UDINT_TO_STRING(ADR(from_rs));
from_rs := SysMemAllocData(name, size*SIZEOF(IP_Buffer), ADR(result));
IF (from_ip = 0) OR (from_rs = 0) THEN
	Init := FALSE;
	fb_exit(FALSE);
	RETURN;
END_IF
SysMemSet(from_ip, 0, size*SIZEOF(IP_Buffer));
SysMemSet(from_rs, 0, size*SIZEOF(IP_Buffer));

FOR i := 0 TO size - 1 DO	
	j := 0;
	msg_qnt := 0;
	WHILE (LEN(clientsCfg[j].client_address) > 0) DO		
		IF (clientsCfg[j].rs_port = portsCfg[i].number) THEN
			msg_qnt := msg_qnt +1;
		END_IF
		j := j+1;
	END_WHILE
	IF (msg_qnt <> 0) THEN		
		from_ip[i].size := msg_qnt*2;
		name := UDINT_TO_STRING(ADR(from_ip[i]));
		from_ip[i].messages := SysMemAllocData(name, from_ip[i].size*SIZEOF(IP_Message), ADR(result));
		from_rs[i].size := msg_qnt*4;
		name := UDINT_TO_STRING(ADR(from_rs[i]));
		from_rs[i].messages := SysMemAllocData(name, from_rs[i].size*SIZEOF(IP_Message), ADR(result));
		IF (from_ip[i].messages = 0) OR (from_rs[i].messages = 0) THEN
			Init := FALSE;
			fb_exit(FALSE);
			RETURN;
		END_IF
		SysMemSet(from_ip[i].messages, 0, from_ip[i].size*SIZEOF(IP_Message));
		SysMemSet(from_rs[i].messages, 0, from_rs[i].size*SIZEOF(IP_Message));
		from_ip[i].rs_port := portsCfg[i].number;
		from_rs[i].rs_port := portsCfg[i].number;
	END_IF	
END_FOR

Init := TRUE;
END_METHOD

METHOD GetMessageForIP : BOOL
VAR_INPUT
	ip_port			: UINT;
	address			: UDINT;
	rs_port			: UINT;
	state			: POINTER TO UINT;
	data			: POINTER TO BYTE;
	size			: UINT;
	length			: POINTER TO UINT;	
END_VAR
VAR
	i				: UINT;
	local_begin		: UINT;
	local_qnt		: UINT;
	msg				: POINTER TO IP_Message;
END_VAR

GetMessageForIP := FALSE;

IF (from_rs = 0) OR (state = 0) OR (data = 0) OR (length = 0) THEN
	RETURN;
END_IF

FOR i := 0 TO THIS^.size - 1 DO	
	IF (from_rs[i].rs_port = rs_port) AND (from_rs[i].size <> 0) THEN	
		local_begin := from_rs[i].begin;
		local_qnt := from_rs[i].qnt;
		WHILE (local_qnt <> 0) DO
			msg := ADR(from_rs[i].messages[local_begin]);			
			IF (msg^.ip_port = ip_port) AND (msg^.address = address) THEN
				IF (msg^.length <= size) THEN				
					state^ := msg^.state;
					SysMemCpy(data, ADR(msg^.data), msg^.length);
					length^ := msg^.length;					
					DeleteMessage(ADR(from_rs[i]), local_begin);
					GetMessageForIP := TRUE;
					RETURN;
				ELSE
					DeleteMessage(ADR(from_rs[i]), local_begin);					
				END_IF;
			END_IF			
			local_begin := (local_begin + 1) MOD from_rs[i].size;
			local_qnt := local_qnt - 1;
		END_WHILE
	END_IF
END_FOR
END_METHOD

METHOD DeleteMessage
VAR_INPUT
	buffer			: POINTER TO IP_Buffer;
	msg_index		: UINT;
END_VAR
VAR
	i_to, i_from	: UINT;
END_VAR
IF (buffer = 0) OR (buffer^.qnt = 0) OR (msg_index >= buffer^.size) THEN
	RETURN;
END_IF

i_to := msg_index;
WHILE (i_to <> buffer^.begin) DO	
	IF (i_to > 0) THEN
		i_from := i_to - 1;			
	ELSE
		i_from := buffer^.size - 1;
	END_IF		
	SysMemCpy(ADR(buffer^.messages[i_to]), ADR(buffer^.messages[i_from]), SIZEOF(IP_Message));
	i_to := i_from;
END_WHILE

buffer^.qnt := buffer^.qnt - 1;
buffer^.begin := (buffer^.begin + 1) MOD buffer^.size;
END_METHOD

METHOD fb_exit : BOOL
VAR_INPUT
	bInCopyCode : BOOL; // if TRUE, the exit method is called for exiting an instance that is copied afterwards (online change). 
END_VAR
VAR
	i		: UINT;
	name	: string;
END_VAR

IF (from_ip <> 0) THEN
	FOR i := 0 TO size - 1 DO	
		IF (from_ip[i].messages <> 0) THEN
			name := UDINT_TO_STRING(ADR(from_ip[i]));
			SysMemFreeData(name, from_ip[i].messages);
			from_ip[i].messages := 0;
		END_IF
	END_FOR
	name := UDINT_TO_STRING(THIS);
	SysMemFreeData(name, from_ip);
	from_ip := 0;
END_IF

IF (from_rs <> 0) THEN
	FOR i := 0 TO size - 1 DO	
		IF (from_rs[i].messages <> 0) THEN
			name := UDINT_TO_STRING(ADR(from_rs[i]));
			SysMemFreeData(name, from_rs[i].messages);
			from_rs[i].messages := 0;
		END_IF
	END_FOR
	name := UDINT_TO_STRING(THIS);
	SysMemFreeData(name, from_rs);
	from_rs := 0;
END_IF
END_METHOD

END_FUNCTION_BLOCK

// Serial_port/Serial_group

FUNCTION_BLOCK Serial_group
VAR_INPUT
END_VAR
VAR
	ports			: POINTER TO Serial;	
	ports_qnt		: UINT;
	i				: UINT;
END_VAR

IF (ports = 0) THEN
	RETURN;
END_IF

FOR i := 0 TO ports_qnt - 1 DO
	CASE (ports[i].mode) OF
	SerialConst.HALF_MASTER:
		MasterRun(ADR(ports[i]));	
	SerialConst.HALF_SLAVE:
		SlaveRun(ADR(ports[i]));	
	END_CASE
END_FOR

METHOD SlaveRun
VAR_INPUT
	port				: POINTER TO Serial;
END_VAR
VAR
	comResult			: RTS_IEC_RESULT;
	rx_frame			: ARRAY [0..255] OF BYTE;
	written				: UDINT;
	read				: UDINT;
	tx_attempts			: UDINT;
	ticks				: UDINT;
END_VAR
IF (port = 0) THEN
	RETURN;
END_IF

IF (port^.state = SerialState.INIT)	THEN

	port^.comHandle := SysComOpen2(ADR(port^.settings), 0, ADR(comResult));		
	IF (port^.comHandle = 0) OR (comResult <> CmpErrors.Errors.ERR_OK) THEN
		port^.state := SerialState.ERROR;
	ELSE 
		port^.tx_ip_length := 0;
		port^.wait_start := TRUE;
		port^.state := SerialState.READ;
	END_IF
END_IF		
IF (port^.state = SerialState.START) THEN

	FillTxFrame(port);
	port^.state := SerialState.WRITE;
END_IF			
IF (port^.state = SerialState.WRITE) THEN
		
	written := SysComWrite(port^.comHandle, ADR(port^.tx_frame), port^.tx_frame_len, 0, ADR(comResult));
	
	IF (comResult = CmpErrors.Errors.ERR_OK) THEN
		port^.state := SerialState.READ;	
	ELSIF (comResult = CmpErrors.Errors.ERR_PENDING) THEN
		tx_attempts := tx_attempts + 1;				
	ELSE
		port^.state := SerialState.ERROR;	
	END_IF
END_IF			
IF (port^.state = SerialState.READ) THEN
			
	read := SysComRead(port^.comHandle, ADR(rx_frame[0]), SIZEOF(rx_frame), 0, ADR(comResult));
	
	IF (read <> 0) AND (comResult = CmpErrors.Errors.ERR_OK) THEN
		port^.state := SlaveProcessRx(port, ADR(rx_frame[0]), UDINT_TO_UINT(read));
	ELSIF (comResult <> CmpErrors.Errors.ERR_TIMEOUT) AND (comResult <> CmpErrors.Errors.ERR_PENDING) THEN
		port^.state := SerialState.ERROR;	
	END_IF
END_IF	
IF (port^.state = SerialState.ERROR) THEN
		
	IF (port^.comHandle <> 0) THEN
		comResult := SysComClose(port^.comHandle);			 
	END_IF
	port^.state := SerialState.INIT;
END_IF
END_METHOD

METHOD fb_exit
VAR_INPUT
	bInCopyCode : BOOL; // if TRUE, the exit method is called for exiting an instance that is copied afterwards (online change). 
END_VAR
VAR
	i		: UINT;
	name	: STRING;
END_VAR

IF (ports = 0) THEN
	RETURN;
END_IF

FOR i := 0 TO ports_qnt - 1 DO
	IF (ports[i].comHandle <> 0) THEN
		SysComClose(ports[i].comHandle);			 
	END_IF
END_FOR

name := UDINT_TO_STRING(THIS);
SysMemFreeData(name, ports);
ports := 0;
END_METHOD

METHOD fb_init : BOOL
VAR_INPUT
	bInitRetains	: BOOL; // if TRUE, the retain variables are initialized (warm start / cold start)
	bInCopyCode		: BOOL;  // if TRUE, the instance afterwards gets moved into the copy code (online change)
	
	//portsCfg		: POINTER TO SerialCfg;
	//	: POINTER TO Exchange_Buffer;
END_VAR
VAR
	i			: UINT;
	result		: RTS_IEC_RESULT;
	name		: STRING;
END_VAR
(*
ports := 0;

IF (portsCfg = 0) OR (ip2rs_buffer = 0) THEN
	fb_init := FALSE;
	RETURN;
END_IF

i := 0;
WHILE (portsCfg[i].number > 0) DO
	i := i+1;
END_WHILE

IF i = 0 THEN
	fb_init := FALSE;
	RETURN;
END_IF

ports_qnt := i;
name := UDINT_TO_STRING(THIS);
ports := SysMemAllocData(name, ports_qnt*SIZEOF(Serial), ADR(result));
IF ports = 0 THEN
	fb_init := FALSE;
	RETURN;
END_IF

SysMemSet(ports, 0, ports_qnt*SIZEOF(Serial));
FOR i := 0 TO ports_qnt - 1 DO
	ports[i].buffer := ip2rs_buffer;
	ports[i].mode := portsCfg[i].mode;	
	ports[i].settings.byParity := portsCfg[i].parity;
	ports[i].settings.sPort := portsCfg[i].number;
	ports[i].settings.ulBaudrate := portsCfg[i].baudrate;
	ports[i].settings.byStopBits := portsCfg[i].stopbits;
	ports[i].settings.ulBufferSize := portsCfg[i].frame_size;
	ports[i].settings.ulTimeout := portsCfg[i].timeout;
	
	ports[i].timeout := 3000;
	ports[i].attempts := 3;
	
END_FOR

fb_init := TRUE;
*)
END_METHOD

METHOD MasterRun
VAR_INPUT
	port				: POINTER TO Serial;
END_VAR
VAR
	comResult			: RTS_IEC_RESULT;
	rx_frame			: ARRAY [0..255] OF BYTE;
	written				: UDINT;
	read				: UDINT;
	tx_attempts			: UDINT;
	ticks				: UDINT;
END_VAR
IF (port = 0) THEN
	RETURN;
END_IF

IF (port^.state = SerialState.INIT)	THEN

	port^.comHandle := SysComOpen2(ADR(port^.settings), 0, ADR(comResult));		
	IF (port^.comHandle = 0) OR (comResult <> CmpErrors.Errors.ERR_OK) THEN
		port^.state := SerialState.ERROR;
	ELSE
		port^.tx_seq := 1;			
		port^.tx_ip_length := 0;
		port^.wait_start := TRUE;
		port^.state := SerialState.START;
	END_IF
END_IF
IF (port^.state = SerialState.START) THEN

	FillTxFrame(port);
	port^.state := SerialState.WRITE;
	port^.write_attempts := port^.attempts;
END_IF
IF (port^.state = SerialState.WRITE) THEN	
		
	written := SysComWrite(port^.comHandle, ADR(port^.tx_frame), port^.tx_frame_len, 0, ADR(comResult));
	
	IF (comResult = CmpErrors.Errors.ERR_OK) THEN
		port^.state := SerialState.READ;
		port^.write_ticks := SysTimeGetMs();		
	ELSIF (comResult = CmpErrors.Errors.ERR_PENDING) THEN
		tx_attempts := tx_attempts + 1;				
	ELSE
		port^.state := SerialState.ERROR;	
	END_IF
END_IF			
IF (port^.state = SerialState.READ) THEN
			
	read := SysComRead(port^.comHandle, ADR(rx_frame[0]), SIZEOF(rx_frame), 0, ADR(comResult));
	
	IF (read <> 0) AND (comResult = CmpErrors.Errors.ERR_OK) THEN
		IF (MasterProcessRx(port, ADR(rx_frame[0]), UDINT_TO_UINT(read))) THEN
			port^.state := SerialState.START;				
		ELSIF (port^.write_attempts > 0) THEN
			port^.write_attempts := port^.write_attempts - 1;
			port^.state := SerialState.WRITE;
		ELSE
			port^.tx_ip_length := 0;					
			port^.state := SerialState.START;
		END_IF
	ELSIF (comResult = CmpErrors.Errors.ERR_TIMEOUT) OR (comResult = CmpErrors.Errors.ERR_PENDING) THEN
		ticks := SysTimeGetMs() - port^.write_ticks;
		IF (ticks > port^.timeout) THEN				
			IF (port^.write_attempts > 0) THEN
				port^.write_attempts := port^.write_attempts - 1;
				port^.state := SerialState.WRITE;
			ELSE
				port^.tx_ip_length := 0;
				port^.state := SerialState.START;
			END_IF				
		END_IF		
	ELSE
		port^.state := SerialState.ERROR;	
	END_IF
END_IF	
IF (port^.state = SerialState.ERROR) THEN
		
	IF (port^.comHandle <> 0) THEN
		comResult := SysComClose(port^.comHandle);			 
	END_IF
	port^.state := SerialState.INIT;
END_IF
END_METHOD

METHOD SlaveProcessRx : SerialState
VAR_INPUT
	port			: POINTER TO Serial;
	data			: POINTER TO BYTE;
	size			: UINT;
END_VAR
VAR
	header			: POINTER TO SerialHeader;
	max_length		: BYTE;
	length			: UINT;
	crc16			: UINT;
END_VAR
SlaveProcessRx := SerialState.READ;

IF (port = 0) OR (data = 0) OR (size < SIZEOF(SerialHeader) + SIZEOF(crc16)) THEN
	RETURN;
END_IF

header := data;
crc16 :=  MEM.CRC16_Modbus(data, size);
IF (crc16 <> 0) OR (data[0] <> SerialConst.START_BYTE) OR (size <> header^.length + SIZEOF(SerialHeader) + SIZEOF(crc16)) THEN
	RETURN;
END_IF

IF (port^.rx_seq = header^.tx_seq) THEN
	IF (port^.tx_frame_len <> 0) THEN
		SlaveProcessRx := SerialState.WRITE;
	END_IF
	RETURN;
END_IF

IF (port^.rx_seq + 1 <> header^.tx_seq) THEN
	port^.tx_ip_length := 0;
	port^.wait_start := TRUE;
END_IF		

port^.rx_seq := header^.tx_seq;

IF (header^.flags.2 = 1) THEN
	SlaveProcessRx := SerialState.START;
	RETURN;
END_IF

IF (header^.flags.0 = 1) THEN
	SysMemSet(ADR(port^.rx_ip[0]), 0, SIZEOF(port^.rx_ip));		// пришла первая часть данных
	port^.rx_ip_offset := 0;
	port^.rx_ip_length := 0;
	port^.wait_start := FALSE;
ELSIF (port^.wait_start) THEN
	SlaveProcessRx := SerialState.READ;
	RETURN;	
END_IF

SysMemCpy(ADR(port^.rx_ip[port^.rx_ip_offset]), ADR(data[SIZEOF(SerialHeader)]), header^.length);
port^.rx_ip_offset := port^.rx_ip_offset + header^.length;

IF (header^.flags.1 = 1) THEN
	port^.rx_ip_length := port^.rx_ip_offset;		// пришла последняя часть данных	
	port^.buffer^.AddRSMessage(port^.settings.sPort, ADR(port^.rx_ip[0]), port^.rx_ip_length);
	port^.wait_start := TRUE;
END_IF

SlaveProcessRx := SerialState.START;
END_METHOD

METHOD Init : BOOL
VAR_INPUT
	portsCfg		: POINTER TO SerialCfg;
	ip2rs_buffer	: POINTER TO Exchange_Buffer;
END_VAR
VAR
	i			: UINT;
	result		: RTS_IEC_RESULT;
	name		: STRING;
END_VAR

ports := 0;

IF (portsCfg = 0) OR (ip2rs_buffer = 0) THEN
	Init := FALSE;
	RETURN;
END_IF

i := 0;
WHILE (portsCfg[i].number > 0) DO
	i := i+1;
END_WHILE

IF i = 0 THEN
	Init := FALSE;
	RETURN;
END_IF

ports_qnt := i;
name := UDINT_TO_STRING(THIS);
ports := SysMemAllocData(name, ports_qnt*SIZEOF(Serial), ADR(result));
IF ports = 0 THEN
	Init := FALSE;
	RETURN;
END_IF

SysMemSet(ports, 0, ports_qnt*SIZEOF(Serial));
FOR i := 0 TO ports_qnt - 1 DO
	ports[i].buffer := ip2rs_buffer;
	ports[i].mode := portsCfg[i].mode;	
	ports[i].settings.byParity := portsCfg[i].parity;
	ports[i].settings.sPort := portsCfg[i].number;
	ports[i].settings.ulBaudrate := portsCfg[i].baudrate;
	ports[i].settings.byStopBits := portsCfg[i].stopbits;
	ports[i].settings.ulBufferSize := portsCfg[i].frame_size;
	ports[i].settings.ulTimeout := portsCfg[i].timeout;
	
	ports[i].timeout := 10000;
	ports[i].attempts := 3;
	
END_FOR

Init := TRUE;
END_METHOD

METHOD MasterProcessRx : BOOL
VAR_INPUT
	port			: POINTER TO Serial;
	data			: POINTER TO BYTE;
	size			: UINT;
END_VAR
VAR
	header			: POINTER TO SerialHeader;
	max_length		: BYTE;
	length			: UINT;
	crc16			: UINT;
END_VAR
MasterProcessRx := FALSE;

IF (port = 0) OR (data = 0) OR (size < SIZEOF(SerialHeader) + SIZEOF(crc16)) THEN
	RETURN;
END_IF

header := data;
crc16 :=  MEM.CRC16_Modbus(data, size);
IF (crc16 <> 0) OR (data[0] <> SerialConst.START_BYTE) OR (size <> header^.length + SIZEOF(SerialHeader) + SIZEOF(crc16)) THEN
	RETURN;
END_IF

IF (port^.tx_seq <> header^.rx_seq) THEN
	RETURN;
END_IF

port^.rx_seq := header^.tx_seq;

IF (header^.flags.2 = 1) THEN
	MasterProcessRx := TRUE;
	RETURN;
END_IF

IF (header^.flags.0 = 1) THEN
	SysMemSet(ADR(port^.rx_ip[0]), 0, SIZEOF(port^.rx_ip));		// пришла первая часть данных
	port^.rx_ip_offset := 0;
	port^.rx_ip_length := 0;
	port^.wait_start := FALSE;
ELSIF (port^.wait_start) THEN
	RETURN;	
END_IF

SysMemCpy(ADR(port^.rx_ip[port^.rx_ip_offset]), ADR(data[SIZEOF(SerialHeader)]), header^.length);
port^.rx_ip_offset := port^.rx_ip_offset + header^.length;

IF (header^.flags.1 = 1) THEN
	port^.rx_ip_length := port^.rx_ip_offset;		// пришла последняя часть данных	
	port^.buffer^.AddRSMessage(port^.settings.sPort, ADR(port^.rx_ip[0]), port^.rx_ip_length);
	port^.wait_start := TRUE;
END_IF

MasterProcessRx := TRUE;
END_METHOD

METHOD FillTxFrame
VAR_INPUT
	port			: POINTER TO Serial;	
END_VAR
VAR
	header			: POINTER TO SerialHeader;
	max_length		: UINT;
	length			: UINT;
	crc16			: UINT;
	ip_data			: BOOL;
END_VAR

IF (port = 0) THEN
	RETURN;
END_IF

port^.tx_seq := port^.tx_seq + 1;

header := ADR(port^.tx_frame[0]);		
header^.start := SerialConst.START_BYTE;
header^.flags := 0;
header^.tx_seq := port^.tx_seq;
header^.rx_seq := port^.rx_seq;

IF (port^.tx_ip_length = 0) THEN
	ip_data := port^.buffer^.GetMessageForRS(port^.settings.sPort, ADR(port^.tx_ip[0]), SIZEOF(port^.tx_ip), ADR(port^.tx_ip_length));
	IF (ip_data = FALSE) THEN
		header^.flags.2 := 1;		// передача тестового пакета
		header^.length := 0;		
		port^.tx_frame_len := UDINT_TO_UINT(SIZEOF(SerialHeader));
		crc16 := MEM.CRC16_Modbus(ADR(port^.tx_frame[0]), port^.tx_frame_len);
	//	crc16 := MEM.ReverseBYTEsInWORD(crc16);
		SysMemCpy(ADR(port^.tx_frame[port^.tx_frame_len]), ADR(crc16), SIZEOF(crc16));
		port^.tx_frame_len := port^.tx_frame_len + SIZEOF(crc16);	
		RETURN;
	ELSE
		port^.tx_ip_offset := 0;
		header^.flags.0 := 1;		// передача первой части данных
	END_IF
END_IF;

max_length := UDINT_TO_UINT(port^.settings.ulBufferSize - SIZEOF(SerialHeader) - SIZEOF(crc16));
length := port^.tx_ip_length - port^.tx_ip_offset;

IF (length > max_length) THEN	
	header^.length := UINT_TO_BYTE(max_length);
ELSE
	header^.length := UINT_TO_BYTE(length);	
END_IF

IF (port^.tx_ip_length <= port^.tx_ip_offset + header^.length) THEN	
	header^.flags.1 := 1;		// передача последней части данных
END_IF

port^.tx_frame_len := UDINT_TO_BYTE(SIZEOF(SerialHeader));		
SysMemCpy(ADR(port^.tx_frame[port^.tx_frame_len]), ADR(port^.tx_ip[port^.tx_ip_offset]), header^.length);
port^.tx_frame_len := port^.tx_frame_len + header^.length;	
crc16 :=  MEM.CRC16_Modbus(ADR(port^.tx_frame[0]), port^.tx_frame_len);
//crc16 := MEM.ReverseBYTEsInWORD(crc16);
SysMemCpy(ADR(port^.tx_frame[port^.tx_frame_len]), ADR(crc16), SIZEOF(crc16));
port^.tx_frame_len := port^.tx_frame_len + SIZEOF(crc16);

IF (header^.flags.1 = 1) THEN
	port^.tx_ip_length := 0;
ELSE
	port^.tx_ip_offset := port^.tx_ip_offset + header^.length;
END_IF
END_METHOD

END_FUNCTION_BLOCK

// Client_TCP/Client_group
FUNCTION_BLOCK Client_group
VAR_INPUT
END_VAR
VAR
	clients			: POINTER TO Client;	
	clients_qnt		: UINT;
	i				: UINT;
END_VAR

IF (clients = 0) THEN
	RETURN;
END_IF

FOR i := 0 TO clients_qnt - 1 DO
	ClientRun(ADR(clients[i]));
END_FOR

METHOD Init : BOOL
VAR_INPUT
	clientsCfg		: POINTER TO ClientCfg;
	ip2rs_buffer	: POINTER TO Exchange_Buffer;
END_VAR
VAR
	i			: UINT;
	result		: RTS_IEC_RESULT;
	address		: SOCKADDRESS;
	name		: STRING;
END_VAR
clients := 0;

IF (clientsCfg = 0) OR (ip2rs_buffer = 0) THEN
	Init := FALSE;
	RETURN;
END_IF


i := 0;
WHILE (LEN(clientsCfg[i].client_address)>0) AND (i < CLIENT_MAX_COUNT) DO
	i := i+1;
END_WHILE

IF i = 0 THEN
	Init := FALSE;
	RETURN;
END_IF

clients_qnt := i;
name := UDINT_TO_STRING(THIS);
clients := SysMemAllocData(name, clients_qnt*SIZEOF(Client), ADR(result));
IF clients = 0 THEN
	Init := FALSE;
	RETURN;
END_IF

SysMemSet(clients, 0, clients_qnt*SIZEOF(Client));
FOR i := 0 TO clients_qnt - 1 DO
		
	address.sin_family := SOCKET_AF_INET;
	address.sin_port := SysSockHtons(clientsCfg[i].server_port);
	result := SysSockInetAddr(clientsCfg[i].client_address, ADR(address.sin_addr.ulAddr));
	IF result <> CmpErrors.Errors.ERR_OK THEN
		Init := FALSE;
		fb_exit(FALSE);
		RETURN;
	END_IF	
	clients[i].from_address := address;
	
	address.sin_family := SOCKET_AF_INET;
	address.sin_port := SysSockHtons(clientsCfg[i].route_port);
	result := SysSockInetAddr(clientsCfg[i].route_address, ADR(address.sin_addr.ulAddr));
	IF result <> CmpErrors.Errors.ERR_OK THEN
		Init := FALSE;
		fb_exit(FALSE);
		RETURN;
	END_IF	
	clients[i].to_address := address;
	
	clients[i].rs_port := clientsCfg[i].rs_port;	
	clients[i].buffer := ip2rs_buffer;
END_FOR

Init := TRUE;
END_METHOD

METHOD ClientRun
VAR_INPUT
	cli : POINTER TO Client;
END_VAR
VAR
	result				: RTS_IEC_RESULT;
	client_socket		: SysSocket.RTS_IEC_HANDLE;
	count				: UINT;
	fdRead				: SOCKET_FD_SET;
	fdExcept			: SOCKET_FD_SET;
	timeout				: SOCKET_TIMEVAL;
	diReady				: DINT;	
	numberofbytes		:__XINT;
	tx_length			: UINT;
	need_tx				: BOOL;
	ip_state			: UINT;	
	non_blocking		: DINT := 1;
END_VAR
IF (cli = 0) THEN
	RETURN;
END_IF

IF (cli^.state = ClientState.RUN) THEN
	
	need_tx := cli^.buffer^.GetMessageForIP(cli^.from_address.sin_port, cli^.from_address.sin_addr.ulAddr, cli^.rs_port, ADR(ip_state), ADR(cli^.tx_data), SIZEOF(cli^.tx_data), ADR(tx_length));		
	IF (need_tx) THEN
		CASE (ip_state) OF		
			WORK_CONNECTION:
				IF (cli^.socket <> 0) THEN
					numberofbytes := SysSockSend(cli^.socket, ADR(cli^.tx_data), tx_length, 0, ADR(result));
					IF (result <> CmpErrors.Errors.ERR_OK AND result <> CmpErrors.Errors.ERR_SOCK_WOULDBLOCK) THEN
						ClientClose(cli, FALSE);
					END_IF
				END_IF	
			OPEN_CONNECTION:
				IF (cli^.socket <> 0) THEN
					ClientClose(cli, TRUE);			
				END_IF
				cli^.state := ClientState.CREATE;						
			CLOSE_CONNECTION:
				ClientClose(cli, TRUE);				
			REOPEN_CONNECTION:
				IF (cli^.socket <> 0) THEN
					ClientClose(cli, TRUE);								
				END_IF
				cli^.state := ClientState.CREATE;
		END_CASE
	END_IF
	
	IF (cli^.socket <> 0) THEN

		SysSockFdZero(fdRead);
		SysSockFdZero(fdExcept);		
		count := cli^.buffer^.CheckIPMessage(cli^.from_address.sin_port, cli^.from_address.sin_addr.ulAddr, cli^.rs_port);		
		IF (count = 0) THEN
			SysSockFdInit(cli^.socket, fdRead);
		END_IF
			SysSockFdInit(cli^.socket, fdExcept);

		timeout.tv_sec := 0;
		timeout.tv_usec := 0;
		result := SysSockSelect(1, ADR(fdRead), 0, ADR(fdExcept), ADR(timeout), ADR(diReady));
 
		IF (result <> CmpErrors.Errors.ERR_OK) THEN		
			ClientClose(cli, FALSE);
		ELSIF (diReady <> 0) THEN
			IF SysSockFdIsset(cli^.socket, fdExcept) THEN
				ClientClose(cli, FALSE);
			ELSIF SysSockFdIsset(cli^.socket, fdRead) THEN				
				numberOfBytes := SysSockRecv(cli^.socket, ADR(cli^.rx_data), SIZEOF(cli^.rx_data), 0, ADR(result));	
				IF (result <> CmpErrors.Errors.ERR_OK AND result <> CmpErrors.Errors.ERR_SOCK_WOULDBLOCK) THEN				
					ClientClose(cli, FALSE);		
				ELSIF (numberOfBytes <> 0) THEN
					cli^.buffer^.AddIPMessage(cli^.from_address.sin_port, cli^.from_address.sin_addr.ulAddr, cli^.rs_port, WORK_CONNECTION, ADR(cli^.rx_data), DINT_TO_UINT(numberOfBytes));
				END_IF
			END_IF			
		END_IF
	END_IF
END_IF
IF (cli^.state = ClientState.CREATE) THEN
	
	client_socket := SysSockCreate(SOCKET_AF_INET, SOCKET_STREAM, SOCKET_IPPROTO_TCP, ADR(result));
	IF (client_socket = SysSocket.RTS_INVALID_HANDLE) THEN
		RETURN;	// Fatal Error!!!!  что делать?
	END_IF
	cli^.socket := client_socket;
	result := SysSockIoctl(cli^.socket, SOCKET_FIONBIO, ADR(non_blocking));
	IF result = CmpErrors.Errors.ERR_OK THEN
		cli^.state := ClientState.CONNECT;
	ELSE
		ClientClose(cli, FALSE);
		cli^.state := ClientState.RUN;
	END_IF
END_IF
IF (cli^.state = ClientState.CONNECT) THEN
	
		result := SysSockConnect(cli^.socket, ADR(cli^.to_address), SIZEOF(SOCKADDRESS));		
		IF (result = CmpErrors.Errors.ERR_SOCK_ISCONNECTED) OR (result = CmpErrors.Errors.ERR_OK) THEN		
			cli^.state := ClientState.RUN;
		ELSIF result <> CmpErrors.Errors.ERR_SOCK_WOULDBLOCK THEN
			ClientClose(cli, FALSE);
			cli^.state := ClientState.RUN;
		END_IF 
END_IF
END_METHOD

METHOD ClientClose
VAR_INPUT
	cli			: POINTER TO Client;
	reopen		: BOOL;
END_VAR
VAR
	result				: RTS_IEC_RESULT;
END_VAR
IF (cli = 0) THEN
	RETURN;
END_IF

IF (cli^.socket <> 0) THEN
	result := SysSockClose(cli^.socket);
	cli^.socket := 0;	
	IF (reopen = FALSE) THEN
		cli^.buffer^.ClearByClient(cli^.from_address.sin_port, cli^.from_address.sin_addr.ulAddr, cli^.rs_port);
		cli^.buffer^.AddIPMessage(cli^.from_address.sin_port, cli^.from_address.sin_addr.ulAddr, cli^.rs_port, CLOSE_CONNECTION, ADR(cli^.rx_data), 0);
	END_IF
	cli^.ttl := 0;
END_IF
END_METHOD

METHOD fb_init : BOOL
VAR_INPUT
	bInitRetains : BOOL; // if TRUE, the retain variables are initialized (warm start / cold start)
	bInCopyCode  : BOOL; // if TRUE, the instance afterwards gets moved into the copy code (online change)
END_VAR
END_METHOD

METHOD fb_exit : BOOL
VAR_INPUT
	bInCopyCode : BOOL; // if TRUE, the exit method is called for exiting an instance that is copied afterwards (online change). 
END_VAR
VAR
	i		: UINT;
	result	: RTS_IEC_RESULT;
	name	: STRING;
END_VAR

IF (clients = 0) THEN
	RETURN;
END_IF

FOR i := 0 TO clients_qnt - 1 DO
	IF clients[i].socket <> 0 THEN 
		SysSockClose(clients[i].socket);
		clients[i].socket := 0;
	END_IF;	
END_FOR

name := UDINT_TO_STRING(THIS);
SysMemFreeData(name, clients);
clients := 0;
END_METHOD

END_FUNCTION_BLOCK

// A1_01A/Application/Oscat/T_PLC_US
FUNCTION T_PLC_US : DWORD
VAR CONSTANT
	debug : BOOL := 0;
	N : INT := 0;
	offset : DWORD := 0;
END_VAR
VAR
	tx : TIME;
END_VAR

(*
version 1.2	16 nov 2008
programmer 	hugo
tested by	tobias

T_PLC_US reads the internal PLC timer and return the time, it has the advantage to be able to set a debug mode 
and speed up the counter to test the plc timer overrun which occurs every 50 days respectively 25 days at siemens S7
this routine also allows to correct the behavior of s7 where the internal plc counter will not count all 32 bits.

*)

tx := TIME();
T_PLC_US := TIME_TO_DWORD(Tx)*1000;
(* hier muss die korrektur für step7 stattfinden
plctime muss den vollen wertebereich von time ausnutzen:
wenn bei step7 time -24tage bis plus 24 tage ist dann muss der timer auch beim überlauf auf -24tage springen 
und auf keinen fall auf 0 !!!!
für siemens muss ein weiterer fb im main eingebunden werden der sicherstellt das alle 32 bits durchgezählt werden.
es kann nur ein fb sein den er muss sich das oberste (32te) bit merken.
oder etwa spring s7 bei überlauf auf -24 tage????? dann wäre keine korrektur nötig.
*)
IF debug THEN
	T_PLC_US := (SHL(T_PLC_US,N) OR SHL(DWORD#1,N)-1) + OFFSET;
END_IF;

(* revision history
hm	14.9.2007	rev 1.0
	original version

hm	12. nov 2007	rev 1.1
	added temporaray variable tx because some compilers could not handle time() as an argument

hm	16. nov. 2008	rev 1.2
	initialized constants with 0 for compatibility reasons

*)

END_FUNCTION

// A1_01A/Application/Oscat/CTRL_OUT
FUNCTION_BLOCK CTRL_OUT
VAR_INPUT
	CI, OFFSET, MAN_IN, LIM_L, LIM_H : REAL;
	MANUAL : BOOL;
END_VAR
VAR_OUTPUT
	Y : REAL;
	LIM : BOOL;
END_VAR


(*
version 1.1	5. nov 2008
programmer 	hugo
tested by	oscat


*)

Y := SEL(MANUAL, CI, MAN_IN) + OFFSET;

(* Limit the output *)
IF Y > LIM_L AND Y < LIM_H THEN
	LIM := FALSE;
ELSE
	Y := LIMIT(LIM_L, Y, LIM_H);
	LIM := TRUE;
END_IF;



(* revision history
hm 	2. jun. 2008 	rev 1.0
	original version

hm	5. nov. 2008	rev 1.1
	optimized code
*)

END_FUNCTION_BLOCK

// A1_01A/Application/Oscat/FT_PIDWL
FUNCTION_BLOCK FT_PIDWL
VAR_INPUT
	IN : REAL;
	KP : REAL := 1.0;
	TN : REAL := 1.0;
	TV : REAL := 1.0;
	LIM_L : REAL := -1.0E38;
	LIM_H : REAL := 1.0E38;
	RST : BOOL;
END_VAR
VAR_OUTPUT
	Y : REAL;
	Y_p : REAL;
	Y_i : REAL;
	Y_d : REAL;
	LIM : BOOL;
END_VAR
VAR
	piwl : FT_PIWL;
	diff : FT_DERIV;
END_VAR

(*
version 1.3	13. nov. 2009
programmer 	hugo
tested by		tobias

FT_PIDWL is a PID controller with dynamic wind_up reset.
The PID controller works according to the fomula Y = KP *(IN + KI * INTEG(e) + DERIV(e) ).
a rst will reset the integrator to 0
lim_h and Lim_l set the possible output range of the internal integrator.
the output flags lim will signal that the output limits are active.

default values for KP = 1, KI = 1, ILIM_L = -1E37, iLIM_H = +1E38.
*)

